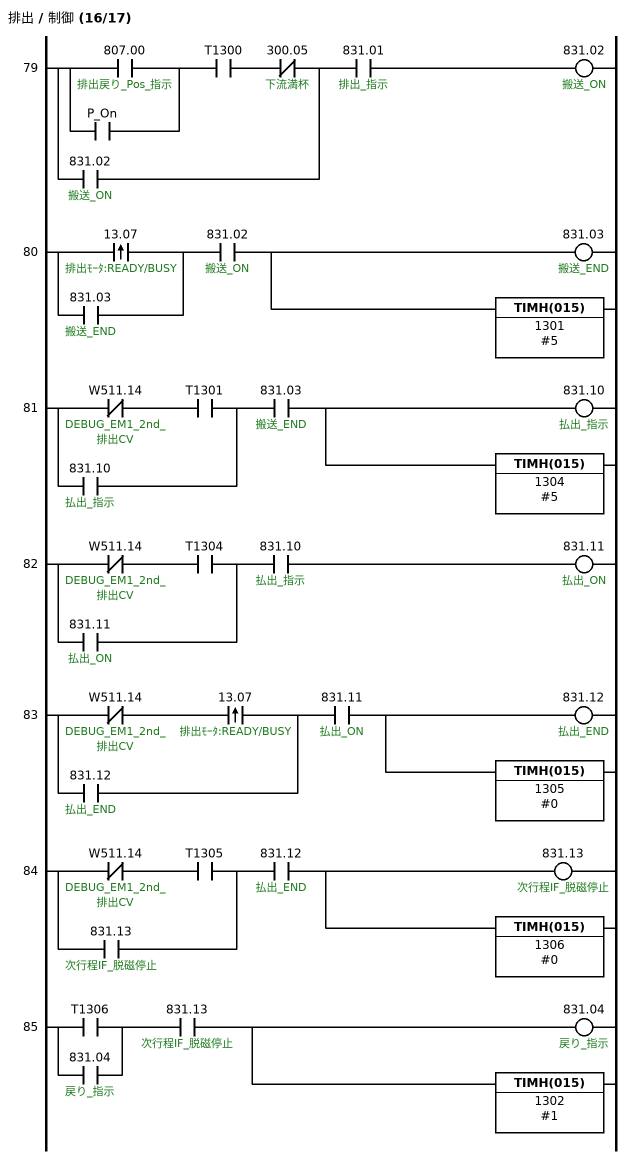
; [picture p192: 排出 / 制御, rungs 79-85]
; rung 79
LD 807.00  ; 排出戻り_Pos_指示
OR P_On
AND T1300
ANDNOT 300.05  ; 下流満杯
OR 831.02  ; 搬送_ON
AND 831.01  ; 排出_指示
OUT 831.02  ; 搬送_ON
; rung 80
@LD 13.07  ; 排出ﾓｰﾀ:READY/BUSY
OR 831.03  ; 搬送_END
AND 831.02  ; 搬送_ON
OUT 831.03  ; 搬送_END
TIMH(015) 1301 #5
; rung 81
LDNOT W511.14  ; DEBUG_EM1_2nd_排出CV
AND T1301
OR 831.10  ; 払出_指示
AND 831.03  ; 搬送_END
OUT 831.10  ; 払出_指示
TIMH(015) 1304 #5
; rung 82
LDNOT W511.14  ; DEBUG_EM1_2nd_排出CV
AND T1304
OR 831.11  ; 払出_ON
AND 831.10  ; 払出_指示
OUT 831.11  ; 払出_ON
; rung 83
LDNOT W511.14  ; DEBUG_EM1_2nd_排出CV
@AND 13.07  ; 排出ﾓｰﾀ:READY/BUSY
OR 831.12  ; 払出_END
AND 831.11  ; 払出_ON
OUT 831.12  ; 払出_END
TIMH(015) 1305 #0
; rung 84
LDNOT W511.14  ; DEBUG_EM1_2nd_排出CV
AND T1305
OR 831.13  ; 次行程IF_脱磁停止
AND 831.12  ; 払出_END
OUT 831.13  ; 次行程IF_脱磁停止
TIMH(015) 1306 #0
; rung 85
LD T1306
OR 831.04  ; 戻り_指示
AND 831.13  ; 次行程IF_脱磁停止
OUT 831.04  ; 戻り_指示
TIMH(015) 1302 #1

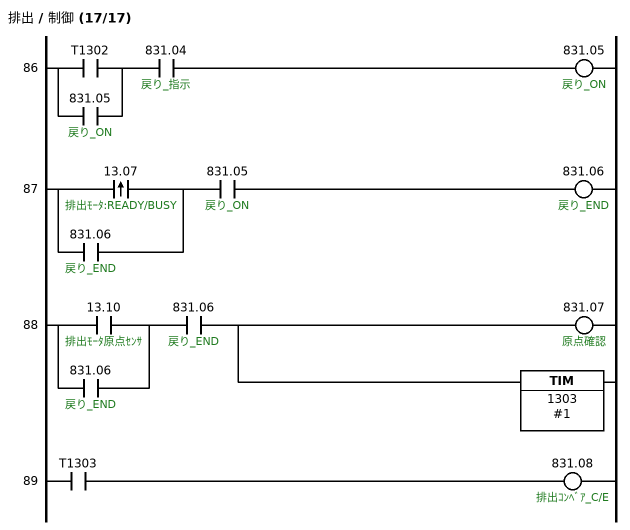
; rung 86
LD T1302
OR 831.05  ; 戻り_ON
AND 831.04  ; 戻り_指示
OUT 831.05  ; 戻り_ON
; rung 87
@LD 13.07  ; 排出ﾓｰﾀ:READY/BUSY
OR 831.06  ; 戻り_END
AND 831.05  ; 戻り_ON
OUT 831.06  ; 戻り_END
; rung 88
LD 13.10  ; 排出ﾓｰﾀ原点ｾﾝｻ
OR 831.06  ; 戻り_END
AND 831.06  ; 戻り_END
OUT 831.07  ; 原点確認
TIM 1303 #1
; rung 89
LD T1303
OUT 831.08  ; 排出ｺﾝﾍﾞｱ_C/E

### Section 出力

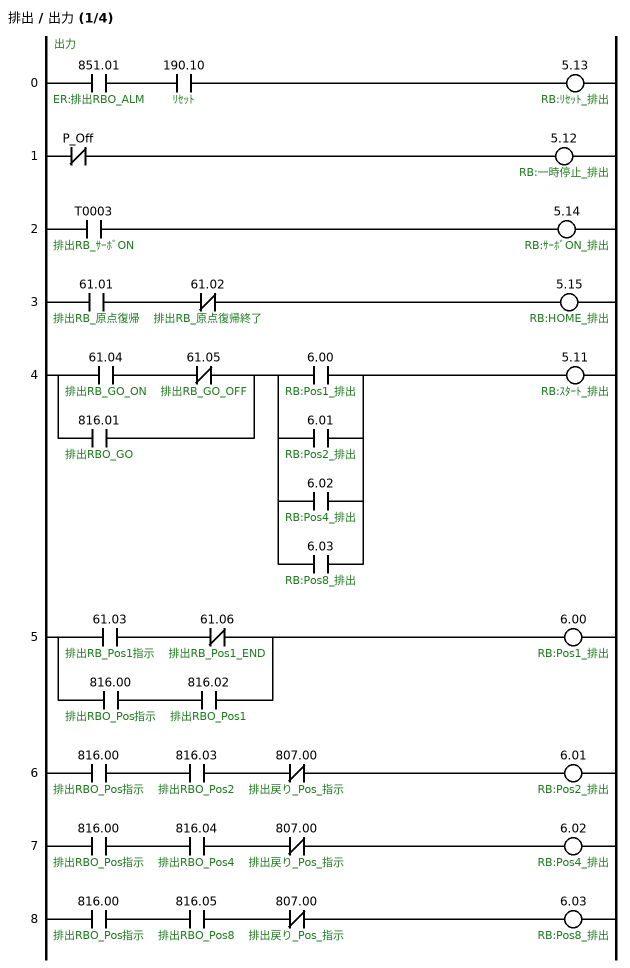
; rung 0: 出力
LD 851.01  ; ER:排出RBO_ALM
AND 190.10  ; ﾘｾｯﾄ
OUT 5.13  ; RB:ﾘｾｯﾄ_排出
; rung 1
LDNOT P_Off
OUT 5.12  ; RB:一時停止_排出
; rung 2
LD T0003  ; 排出RB_ｻｰﾎﾞON
OUT 5.14  ; RB:ｻｰﾎﾞON_排出
; rung 3
LD 61.01  ; 排出RB_原点復帰
ANDNOT 61.02  ; 排出RB_原点復帰終了
OUT 5.15  ; RB:HOME_排出
; rung 4
LD 61.04  ; 排出RB_GO_ON
ANDNOT 61.05  ; 排出RB_GO_OFF
OR 816.01  ; 排出RBO_GO
LD 6.00  ; RB:Pos1_排出
OR 6.01  ; RB:Pos2_排出
OR 6.02  ; RB:Pos4_排出
OR 6.03  ; RB:Pos8_排出
ANDLD
OUT 5.11  ; RB:ｽﾀｰﾄ_排出
; rung 5
LD 61.03  ; 排出RB_Pos1指示
ANDNOT 61.06  ; 排出RB_Pos1_END
LD 816.00  ; 排出RBO_Pos指示
AND 816.02  ; 排出RBO_Pos1
ORLD
OUT 6.00  ; RB:Pos1_排出
; rung 6
LD 816.00  ; 排出RBO_Pos指示
AND 816.03  ; 排出RBO_Pos2
ANDNOT 807.00  ; 排出戻り_Pos_指示
OUT 6.01  ; RB:Pos2_排出
; rung 7
LD 816.00  ; 排出RBO_Pos指示
AND 816.04  ; 排出RBO_Pos4
ANDNOT 807.00  ; 排出戻り_Pos_指示
OUT 6.02  ; RB:Pos4_排出
; rung 8
LD 816.00  ; 排出RBO_Pos指示
AND 816.05  ; 排出RBO_Pos8
ANDNOT 807.00  ; 排出戻り_Pos_指示
OUT 6.03  ; RB:Pos8_排出

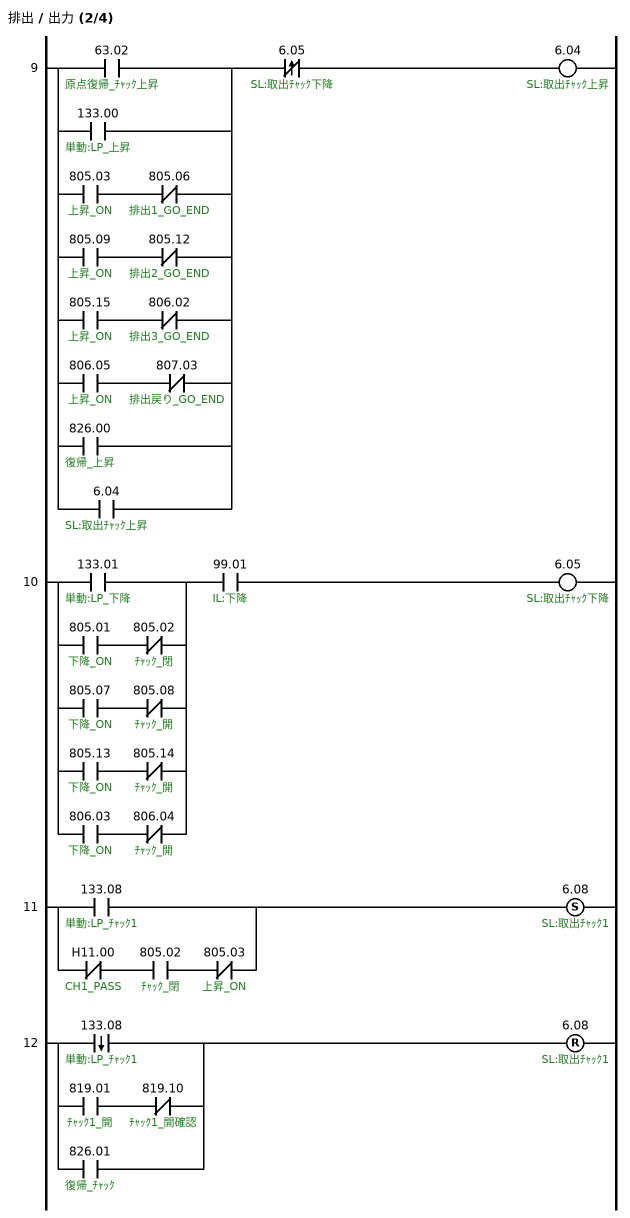
; rung 9
LD 63.02  ; 原点復帰_ﾁｬｯｸ上昇
OR 133.00  ; 単動:LP_上昇
LD 805.03  ; 上昇_ON
ANDNOT 805.06  ; 排出1_GO_END
ORLD
LD 805.09  ; 上昇_ON
ANDNOT 805.12  ; 排出2_GO_END
ORLD
LD 805.15  ; 上昇_ON
ANDNOT 806.02  ; 排出3_GO_END
ORLD
LD 806.05  ; 上昇_ON
ANDNOT 807.03  ; 排出戻り_GO_END
ORLD
OR 826.00  ; 復帰_上昇
OR 6.04  ; SL:取出ﾁｬｯｸ上昇
@ANDNOT 6.05  ; SL:取出ﾁｬｯｸ下降
OUT 6.04  ; SL:取出ﾁｬｯｸ上昇
; rung 10
LD 133.01  ; 単動:LP_下降
LD 805.01  ; 下降_ON
ANDNOT 805.02  ; ﾁｬｯｸ_閉
ORLD
LD 805.07  ; 下降_ON
ANDNOT 805.08  ; ﾁｬｯｸ_開
ORLD
LD 805.13  ; 下降_ON
ANDNOT 805.14  ; ﾁｬｯｸ_開
ORLD
LD 806.03  ; 下降_ON
ANDNOT 806.04  ; ﾁｬｯｸ_開
ORLD
AND 99.01  ; IL:下降
OUT 6.05  ; SL:取出ﾁｬｯｸ下降
; rung 11
LD 133.08  ; 単動:LP_ﾁｬｯｸ1
LDNOT H11.00  ; CH1_PASS
AND 805.02  ; ﾁｬｯｸ_閉
ANDNOT 805.03  ; 上昇_ON
ORLD
SET 6.08  ; SL:取出ﾁｬｯｸ1
; rung 12
%LD 133.08  ; 単動:LP_ﾁｬｯｸ1
LD 819.01  ; ﾁｬｯｸ1_開
ANDNOT 819.10  ; ﾁｬｯｸ1_開確認
ORLD
OR 826.01  ; 復帰_ﾁｬｯｸ
RSET 6.08  ; SL:取出ﾁｬｯｸ1

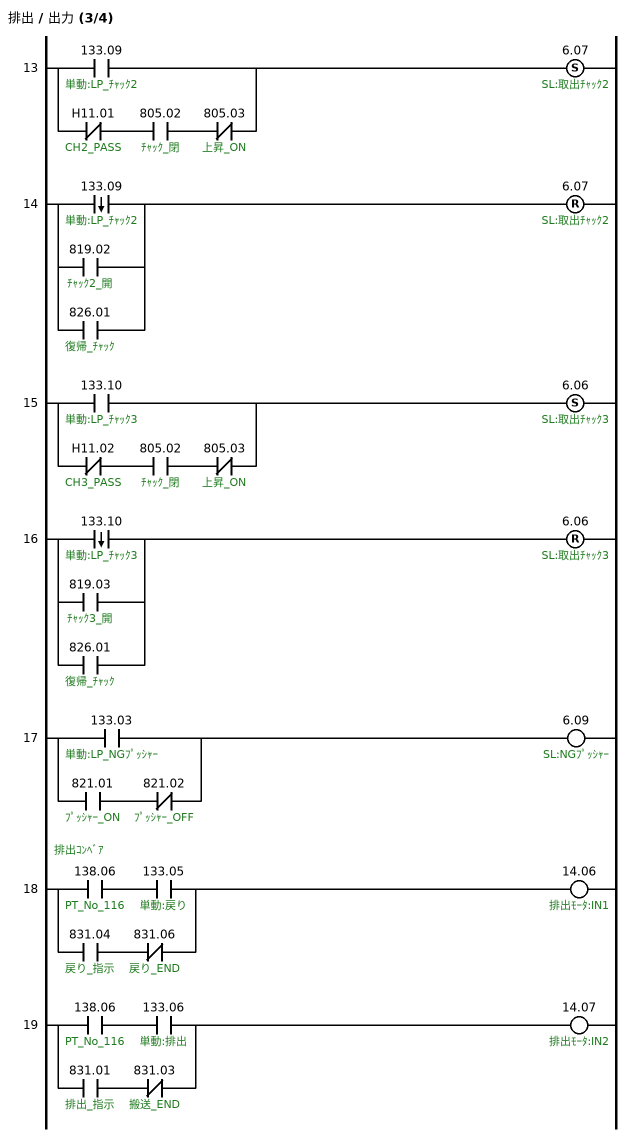
; rung 13
LD 133.09  ; 単動:LP_ﾁｬｯｸ2
LDNOT H11.01  ; CH2_PASS
AND 805.02  ; ﾁｬｯｸ_閉
ANDNOT 805.03  ; 上昇_ON
ORLD
SET 6.07  ; SL:取出ﾁｬｯｸ2
; rung 14
%LD 133.09  ; 単動:LP_ﾁｬｯｸ2
OR 819.02  ; ﾁｬｯｸ2_開
OR 826.01  ; 復帰_ﾁｬｯｸ
RSET 6.07  ; SL:取出ﾁｬｯｸ2
; rung 15
LD 133.10  ; 単動:LP_ﾁｬｯｸ3
LDNOT H11.02  ; CH3_PASS
AND 805.02  ; ﾁｬｯｸ_閉
ANDNOT 805.03  ; 上昇_ON
ORLD
SET 6.06  ; SL:取出ﾁｬｯｸ3
; rung 16
%LD 133.10  ; 単動:LP_ﾁｬｯｸ3
OR 819.03  ; ﾁｬｯｸ3_開
OR 826.01  ; 復帰_ﾁｬｯｸ
RSET 6.06  ; SL:取出ﾁｬｯｸ3
; rung 17
LD 133.03  ; 単動:LP_NGﾌﾟｯｼｬｰ
LD 821.01  ; ﾌﾟｯｼｬｰ_ON
ANDNOT 821.02  ; ﾌﾟｯｼｬｰ_OFF
ORLD
OUT 6.09  ; SL:NGﾌﾟｯｼｬｰ
; rung 18: 排出ｺﾝﾍﾞｱ
LD 138.06  ; PT_No_116
AND 133.05  ; 単動:戻り
LD 831.04  ; 戻り_指示
ANDNOT 831.06  ; 戻り_END
ORLD
OUT 14.06  ; 排出ﾓｰﾀ:IN1  // #1_戻り､#2_排出､#4_払出
; rung 19
LD 138.06  ; PT_No_116
AND 133.06  ; 単動:排出
LD 831.01  ; 排出_指示
ANDNOT 831.03  ; 搬送_END
ORLD
OUT 14.07  ; 排出ﾓｰﾀ:IN2

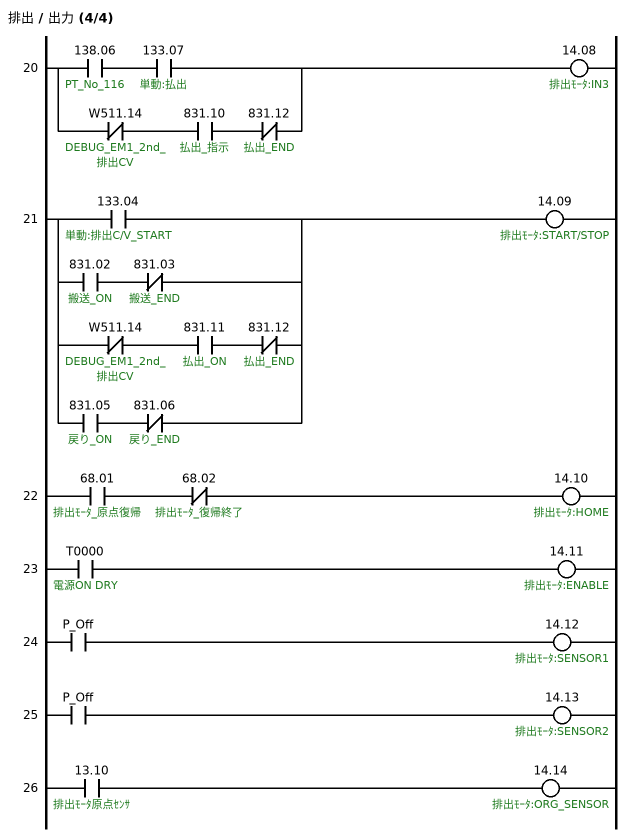
; rung 20
LD 138.06  ; PT_No_116
AND 133.07  ; 単動:払出
LDNOT W511.14  ; DEBUG_EM1_2nd_排出CV
AND 831.10  ; 払出_指示
ANDNOT 831.12  ; 払出_END
ORLD
OUT 14.08  ; 排出ﾓｰﾀ:IN3
; rung 21
LD 133.04  ; 単動:排出C/V_START
LD 831.02  ; 搬送_ON
ANDNOT 831.03  ; 搬送_END
ORLD
LDNOT W511.14  ; DEBUG_EM1_2nd_排出CV
AND 831.11  ; 払出_ON
ANDNOT 831.12  ; 払出_END
ORLD
LD 831.05  ; 戻り_ON
ANDNOT 831.06  ; 戻り_END
ORLD
OUT 14.09  ; 排出ﾓｰﾀ:START/STOP
; rung 22
LD 68.01  ; 排出ﾓｰﾀ_原点復帰
ANDNOT 68.02  ; 排出ﾓｰﾀ_復帰終了
OUT 14.10  ; 排出ﾓｰﾀ:HOME
; rung 23
LD T0000  ; 電源ON DRY
OUT 14.11  ; 排出ﾓｰﾀ:ENABLE
; rung 24
LD P_Off
OUT 14.12  ; 排出ﾓｰﾀ:SENSOR1
; rung 25
LD P_Off
OUT 14.13  ; 排出ﾓｰﾀ:SENSOR2
; rung 26
LD 13.10  ; 排出ﾓｰﾀ原点ｾﾝｻ
OUT 14.14  ; 排出ﾓｰﾀ:ORG_SENSOR

### Section ｴﾗｰ

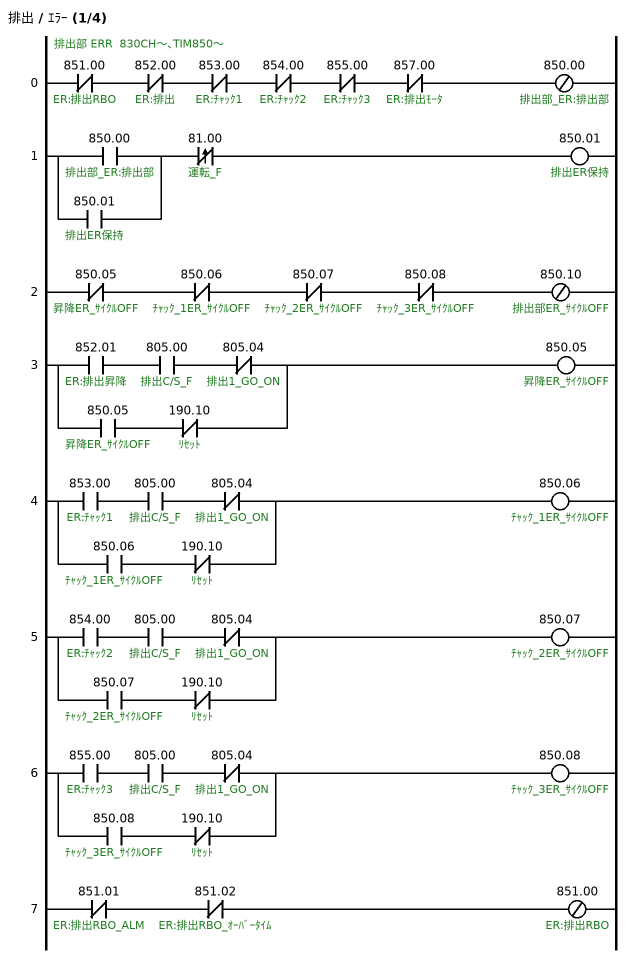
; rung 0: 排出部 ERR  830CH～､TIM850～
LDNOT 851.00  ; ER:排出RBO
ANDNOT 852.00  ; ER:排出
ANDNOT 853.00  ; ER:ﾁｬｯｸ1
ANDNOT 854.00  ; ER:ﾁｬｯｸ2
ANDNOT 855.00  ; ER:ﾁｬｯｸ3
ANDNOT 857.00  ; ER:排出ﾓｰﾀ
OUTNOT 850.00  ; 排出部_ER:排出部
; rung 1
LD 850.00  ; 排出部_ER:排出部
OR 850.01  ; 排出ER保持
@ANDNOT 81.00  ; 運転_F
OUT 850.01  ; 排出ER保持
; rung 2
LDNOT 850.05  ; 昇降ER_ｻｲｸﾙOFF
ANDNOT 850.06  ; ﾁｬｯｸ_1ER_ｻｲｸﾙOFF
ANDNOT 850.07  ; ﾁｬｯｸ_2ER_ｻｲｸﾙOFF
ANDNOT 850.08  ; ﾁｬｯｸ_3ER_ｻｲｸﾙOFF
OUTNOT 850.10  ; 排出部ER_ｻｲｸﾙOFF
; rung 3
LD 852.01  ; ER:排出昇降
AND 805.00  ; 排出C/S_F
ANDNOT 805.04  ; 排出1_GO_ON
LD 850.05  ; 昇降ER_ｻｲｸﾙOFF
ANDNOT 190.10  ; ﾘｾｯﾄ
ORLD
OUT 850.05  ; 昇降ER_ｻｲｸﾙOFF
; rung 4
LD 853.00  ; ER:ﾁｬｯｸ1
AND 805.00  ; 排出C/S_F
ANDNOT 805.04  ; 排出1_GO_ON
LD 850.06  ; ﾁｬｯｸ_1ER_ｻｲｸﾙOFF
ANDNOT 190.10  ; ﾘｾｯﾄ
ORLD
OUT 850.06  ; ﾁｬｯｸ_1ER_ｻｲｸﾙOFF
; rung 5
LD 854.00  ; ER:ﾁｬｯｸ2
AND 805.00  ; 排出C/S_F
ANDNOT 805.04  ; 排出1_GO_ON
LD 850.07  ; ﾁｬｯｸ_2ER_ｻｲｸﾙOFF
ANDNOT 190.10  ; ﾘｾｯﾄ
ORLD
OUT 850.07  ; ﾁｬｯｸ_2ER_ｻｲｸﾙOFF
; rung 6
LD 855.00  ; ER:ﾁｬｯｸ3
AND 805.00  ; 排出C/S_F
ANDNOT 805.04  ; 排出1_GO_ON
LD 850.08  ; ﾁｬｯｸ_3ER_ｻｲｸﾙOFF
ANDNOT 190.10  ; ﾘｾｯﾄ
ORLD
OUT 850.08  ; ﾁｬｯｸ_3ER_ｻｲｸﾙOFF
; rung 7
LDNOT 851.01  ; ER:排出RBO_ALM
ANDNOT 851.02  ; ER:排出RBO_ｵｰﾊﾞｰﾀｲﾑ
OUTNOT 851.00  ; ER:排出RBO

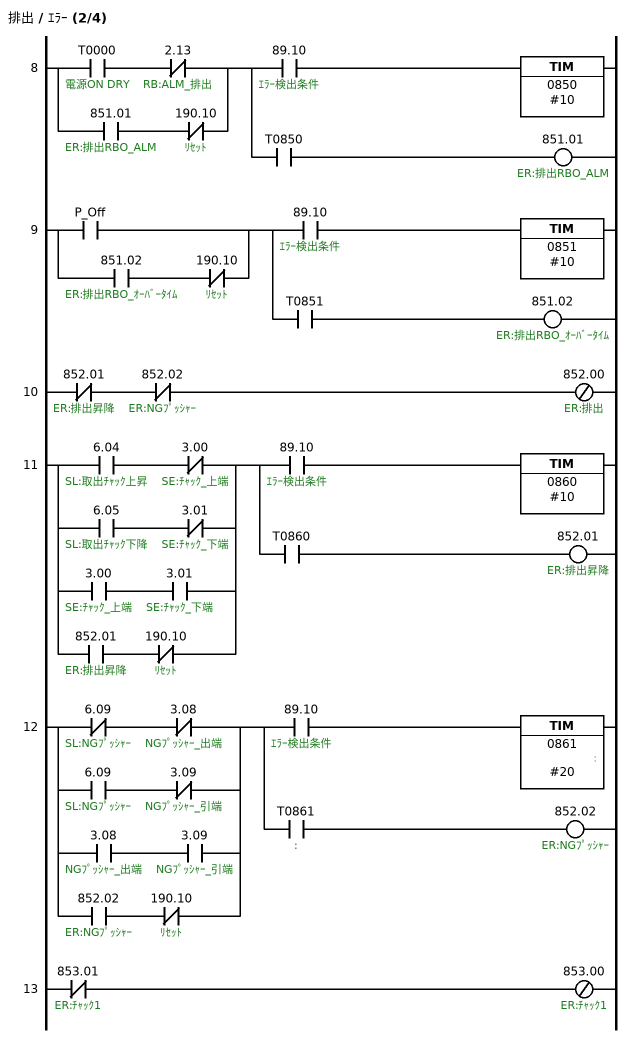
; rung 8
LD T0000  ; 電源ON DRY
ANDNOT 2.13  ; RB:ALM_排出
LD 851.01  ; ER:排出RBO_ALM
ANDNOT 190.10  ; ﾘｾｯﾄ
ORLD
OUT TR0
AND 89.10  ; ｴﾗｰ検出条件
TIM 0850 #10
LD TR0
AND T0850
OUT 851.01  ; ER:排出RBO_ALM
; rung 9
LD P_Off
LD 851.02  ; ER:排出RBO_ｵｰﾊﾞｰﾀｲﾑ
ANDNOT 190.10  ; ﾘｾｯﾄ
ORLD
OUT TR0
AND 89.10  ; ｴﾗｰ検出条件
TIM 0851 #10
LD TR0
AND T0851
OUT 851.02  ; ER:排出RBO_ｵｰﾊﾞｰﾀｲﾑ
; rung 10
LDNOT 852.01  ; ER:排出昇降
ANDNOT 852.02  ; ER:NGﾌﾟｯｼｬｰ
OUTNOT 852.00  ; ER:排出
; rung 11
LD 6.04  ; SL:取出ﾁｬｯｸ上昇
ANDNOT 3.00  ; SE:ﾁｬｯｸ_上端
LD 6.05  ; SL:取出ﾁｬｯｸ下降
ANDNOT 3.01  ; SE:ﾁｬｯｸ_下端
ORLD
LD 3.00  ; SE:ﾁｬｯｸ_上端
AND 3.01  ; SE:ﾁｬｯｸ_下端
ORLD
LD 852.01  ; ER:排出昇降
ANDNOT 190.10  ; ﾘｾｯﾄ
ORLD
OUT TR0
AND 89.10  ; ｴﾗｰ検出条件
TIM 0860 #10
LD TR0
AND T0860
OUT 852.01  ; ER:排出昇降
; rung 12
LDNOT 6.09  ; SL:NGﾌﾟｯｼｬｰ
ANDNOT 3.08  ; NGﾌﾟｯｼｬｰ_出端
LD 6.09  ; SL:NGﾌﾟｯｼｬｰ
ANDNOT 3.09  ; NGﾌﾟｯｼｬｰ_引端
ORLD
LD 3.08  ; NGﾌﾟｯｼｬｰ_出端
AND 3.09  ; NGﾌﾟｯｼｬｰ_引端
ORLD
LD 852.02  ; ER:NGﾌﾟｯｼｬｰ
ANDNOT 190.10  ; ﾘｾｯﾄ
ORLD
OUT TR0
AND 89.10  ; ｴﾗｰ検出条件
TIM 0861 #20  ; :
LD TR0
AND T0861  ; :
OUT 852.02  ; ER:NGﾌﾟｯｼｬｰ
; rung 13
LDNOT 853.01  ; ER:ﾁｬｯｸ1
OUTNOT 853.00  ; ER:ﾁｬｯｸ1

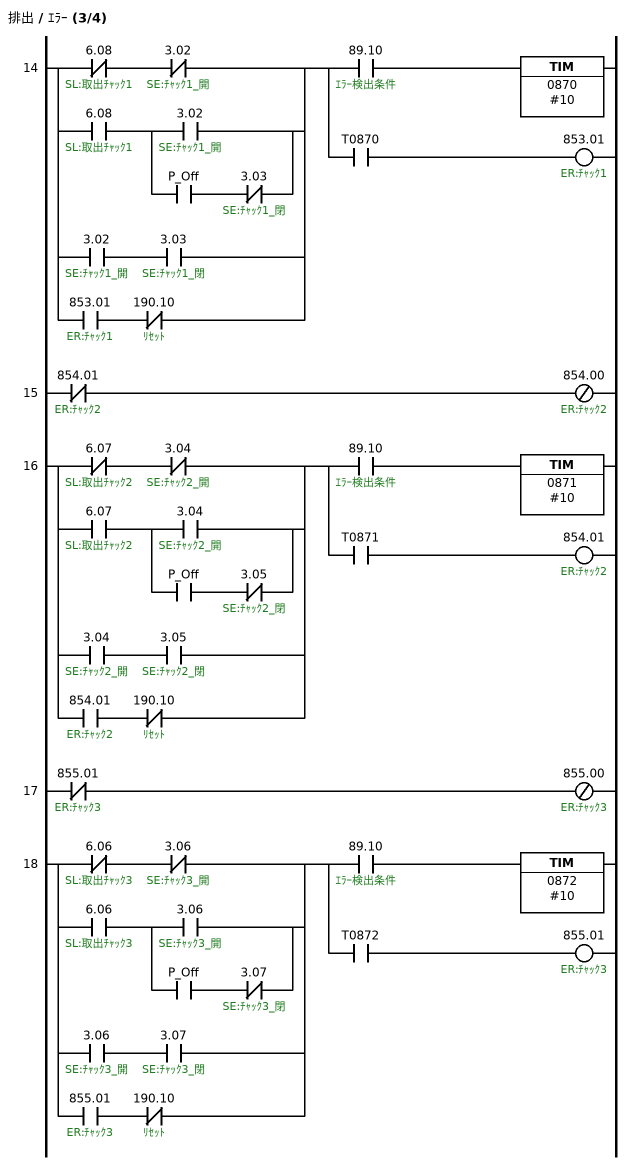
; rung 14
LDNOT 6.08  ; SL:取出ﾁｬｯｸ1
ANDNOT 3.02  ; SE:ﾁｬｯｸ1_開
LD 6.08  ; SL:取出ﾁｬｯｸ1
LD 3.02  ; SE:ﾁｬｯｸ1_開
LD P_Off
ANDNOT 3.03  ; SE:ﾁｬｯｸ1_閉
ORLD
ANDLD
ORLD
LD 3.02  ; SE:ﾁｬｯｸ1_開
AND 3.03  ; SE:ﾁｬｯｸ1_閉
ORLD
LD 853.01  ; ER:ﾁｬｯｸ1
ANDNOT 190.10  ; ﾘｾｯﾄ
ORLD
OUT TR0
AND 89.10  ; ｴﾗｰ検出条件
TIM 0870 #10
LD TR0
AND T0870
OUT 853.01  ; ER:ﾁｬｯｸ1
; rung 15
LDNOT 854.01  ; ER:ﾁｬｯｸ2
OUTNOT 854.00  ; ER:ﾁｬｯｸ2
; rung 16
LDNOT 6.07  ; SL:取出ﾁｬｯｸ2
ANDNOT 3.04  ; SE:ﾁｬｯｸ2_開
LD 6.07  ; SL:取出ﾁｬｯｸ2
LD 3.04  ; SE:ﾁｬｯｸ2_開
LD P_Off
ANDNOT 3.05  ; SE:ﾁｬｯｸ2_閉
ORLD
ANDLD
ORLD
LD 3.04  ; SE:ﾁｬｯｸ2_開
AND 3.05  ; SE:ﾁｬｯｸ2_閉
ORLD
LD 854.01  ; ER:ﾁｬｯｸ2
ANDNOT 190.10  ; ﾘｾｯﾄ
ORLD
OUT TR0
AND 89.10  ; ｴﾗｰ検出条件
TIM 0871 #10
LD TR0
AND T0871
OUT 854.01  ; ER:ﾁｬｯｸ2
; rung 17
LDNOT 855.01  ; ER:ﾁｬｯｸ3
OUTNOT 855.00  ; ER:ﾁｬｯｸ3
; rung 18
LDNOT 6.06  ; SL:取出ﾁｬｯｸ3
ANDNOT 3.06  ; SE:ﾁｬｯｸ3_開
LD 6.06  ; SL:取出ﾁｬｯｸ3
LD 3.06  ; SE:ﾁｬｯｸ3_開
LD P_Off
ANDNOT 3.07  ; SE:ﾁｬｯｸ3_閉
ORLD
ANDLD
ORLD
LD 3.06  ; SE:ﾁｬｯｸ3_開
AND 3.07  ; SE:ﾁｬｯｸ3_閉
ORLD
LD 855.01  ; ER:ﾁｬｯｸ3
ANDNOT 190.10  ; ﾘｾｯﾄ
ORLD
OUT TR0
AND 89.10  ; ｴﾗｰ検出条件
TIM 0872 #10
LD TR0
AND T0872
OUT 855.01  ; ER:ﾁｬｯｸ3

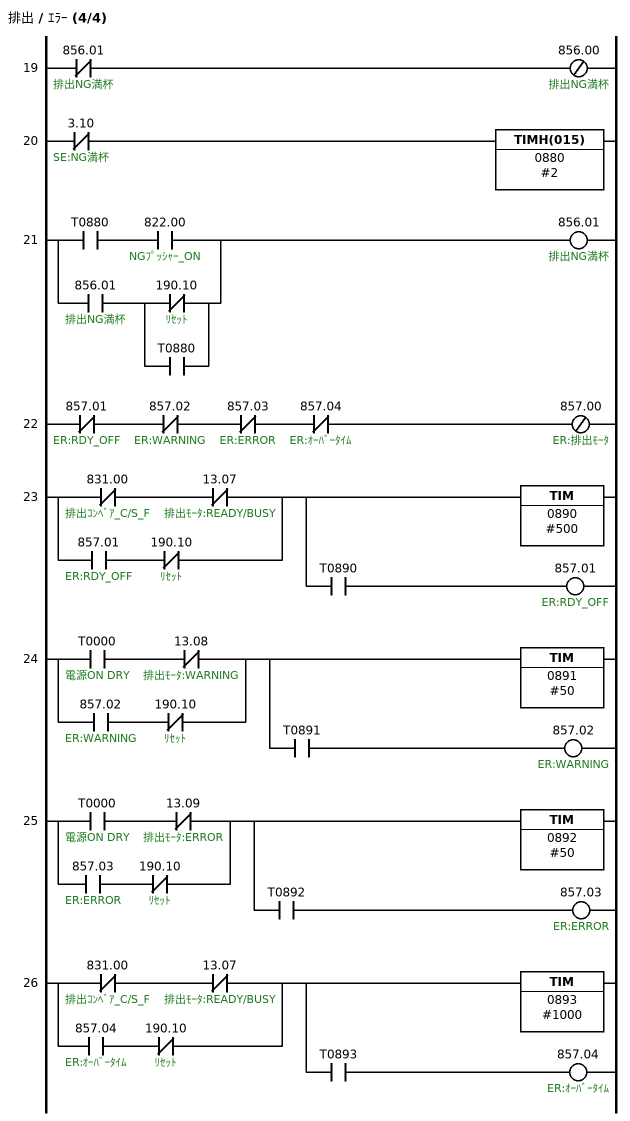
; rung 19
LDNOT 856.01  ; 排出NG満杯
OUTNOT 856.00  ; 排出NG満杯
; rung 20
LDNOT 3.10  ; SE:NG満杯
TIMH(015) 0880 #2
; rung 21
LD T0880
AND 822.00  ; NGﾌﾟｯｼｬｰ_ON
LD 856.01  ; 排出NG満杯
LDNOT 190.10  ; ﾘｾｯﾄ
OR T0880
ANDLD
ORLD
OUT 856.01  ; 排出NG満杯
; rung 22
LDNOT 857.01  ; ER:RDY_OFF
ANDNOT 857.02  ; ER:WARNING
ANDNOT 857.03  ; ER:ERROR
ANDNOT 857.04  ; ER:ｵｰﾊﾞｰﾀｲﾑ
OUTNOT 857.00  ; ER:排出ﾓｰﾀ
; rung 23
LDNOT 831.00  ; 排出ｺﾝﾍﾞｱ_C/S_F
ANDNOT 13.07  ; 排出ﾓｰﾀ:READY/BUSY
LD 857.01  ; ER:RDY_OFF
ANDNOT 190.10  ; ﾘｾｯﾄ
ORLD
TIM 0890 #500
AND T0890
OUT 857.01  ; ER:RDY_OFF
; rung 24
LD T0000  ; 電源ON DRY
ANDNOT 13.08  ; 排出ﾓｰﾀ:WARNING
LD 857.02  ; ER:WARNING
ANDNOT 190.10  ; ﾘｾｯﾄ
ORLD
TIM 0891 #50
AND T0891
OUT 857.02  ; ER:WARNING
; rung 25
LD T0000  ; 電源ON DRY
ANDNOT 13.09  ; 排出ﾓｰﾀ:ERROR
LD 857.03  ; ER:ERROR
ANDNOT 190.10  ; ﾘｾｯﾄ
ORLD
TIM 0892 #50
AND T0892
OUT 857.03  ; ER:ERROR
; rung 26
LDNOT 831.00  ; 排出ｺﾝﾍﾞｱ_C/S_F
ANDNOT 13.07  ; 排出ﾓｰﾀ:READY/BUSY
LD 857.04  ; ER:ｵｰﾊﾞｰﾀｲﾑ
ANDNOT 190.10  ; ﾘｾｯﾄ
ORLD
TIM 0893 #1000
AND T0893
OUT 857.04  ; ER:ｵｰﾊﾞｰﾀｲﾑ

### Section END
; rung 0
END(001)

## Program ﾃﾞｰﾀ収集 (cyclic task 9)

### Section 通信ST

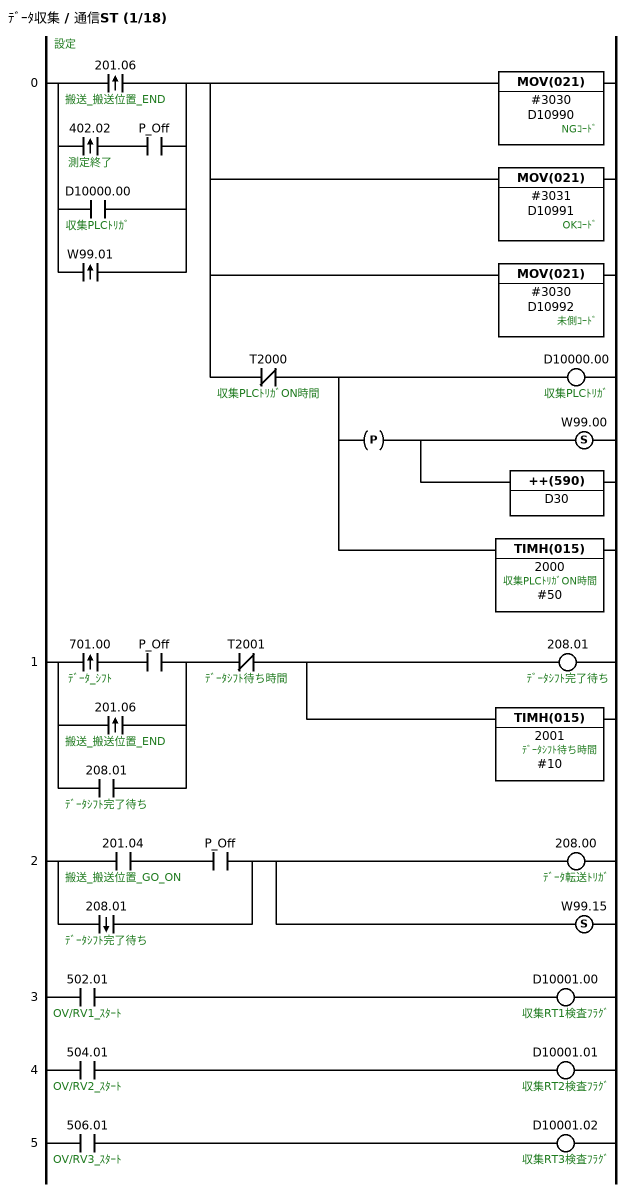
; rung 0: 設定
@LD 201.06  ; 搬送_搬送位置_END
@LD 402.02  ; 測定終了
AND P_Off
ORLD
OR D10000.00  ; 収集PLCﾄﾘｶﾞ
@OR W99.01
MOV(021) #3030 D10990  ; NGｺｰﾄﾞ
MOV(021) #3031 D10991  ; OKｺｰﾄﾞ
MOV(021) #3030 D10992  ; 未側ｺｰﾄﾞ
ANDNOT T2000  ; 収集PLCﾄﾘｶﾞON時間
OUT TR0
OUT D10000.00  ; 収集PLCﾄﾘｶﾞ
UP(521)
SET W99.00
++(590) D30
LD TR0
TIMH(015) 2000 #50  ; 収集PLCﾄﾘｶﾞON時間
; rung 1
@LD 701.00  ; ﾃﾞｰﾀ_ｼﾌﾄ
AND P_Off
@OR 201.06  ; 搬送_搬送位置_END
OR 208.01  ; ﾃﾞｰﾀｼﾌﾄ完了待ち
ANDNOT T2001  ; ﾃﾞｰﾀｼﾌﾄ待ち時間
OUT 208.01  ; ﾃﾞｰﾀｼﾌﾄ完了待ち
TIMH(015) 2001 #10  ; ﾃﾞｰﾀｼﾌﾄ待ち時間
; rung 2
LD 201.04  ; 搬送_搬送位置_GO_ON
AND P_Off
%OR 208.01  ; ﾃﾞｰﾀｼﾌﾄ完了待ち
OUT 208.00  ; ﾃﾞｰﾀ転送ﾄﾘｶﾞ
SET W99.15
; rung 3
LD 502.01  ; OV/RV1_ｽﾀｰﾄ
OUT D10001.00  ; 収集RT1検査ﾌﾗｸﾞ
; rung 4
LD 504.01  ; OV/RV2_ｽﾀｰﾄ
OUT D10001.01  ; 収集RT2検査ﾌﾗｸﾞ
; rung 5
LD 506.01  ; OV/RV3_ｽﾀｰﾄ
OUT D10001.02  ; 収集RT3検査ﾌﾗｸﾞ

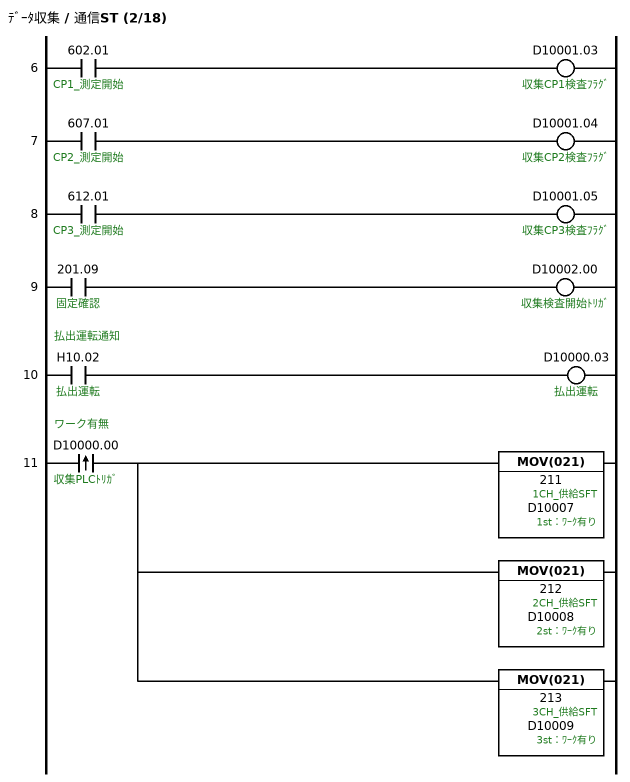
; rung 6
LD 602.01  ; CP1_測定開始
OUT D10001.03  ; 収集CP1検査ﾌﾗｸﾞ
; rung 7
LD 607.01  ; CP2_測定開始
OUT D10001.04  ; 収集CP2検査ﾌﾗｸﾞ
; rung 8
LD 612.01  ; CP3_測定開始
OUT D10001.05  ; 収集CP3検査ﾌﾗｸﾞ
; rung 9
LD 201.09  ; 固定確認
OUT D10002.00  ; 収集検査開始ﾄﾘｶﾞ
; rung 10: 払出運転通知
LD H10.02  ; 払出運転
OUT D10000.03  ; 払出運転
; rung 11: ワーク有無
@LD D10000.00  ; 収集PLCﾄﾘｶﾞ
MOV(021) 211 D10007  ; 1CH_供給SFT, 1st：ﾜｰｸ有り
MOV(021) 212 D10008  ; 2CH_供給SFT, 2st：ﾜｰｸ有り
MOV(021) 213 D10009  ; 3CH_供給SFT, 3st：ﾜｰｸ有り

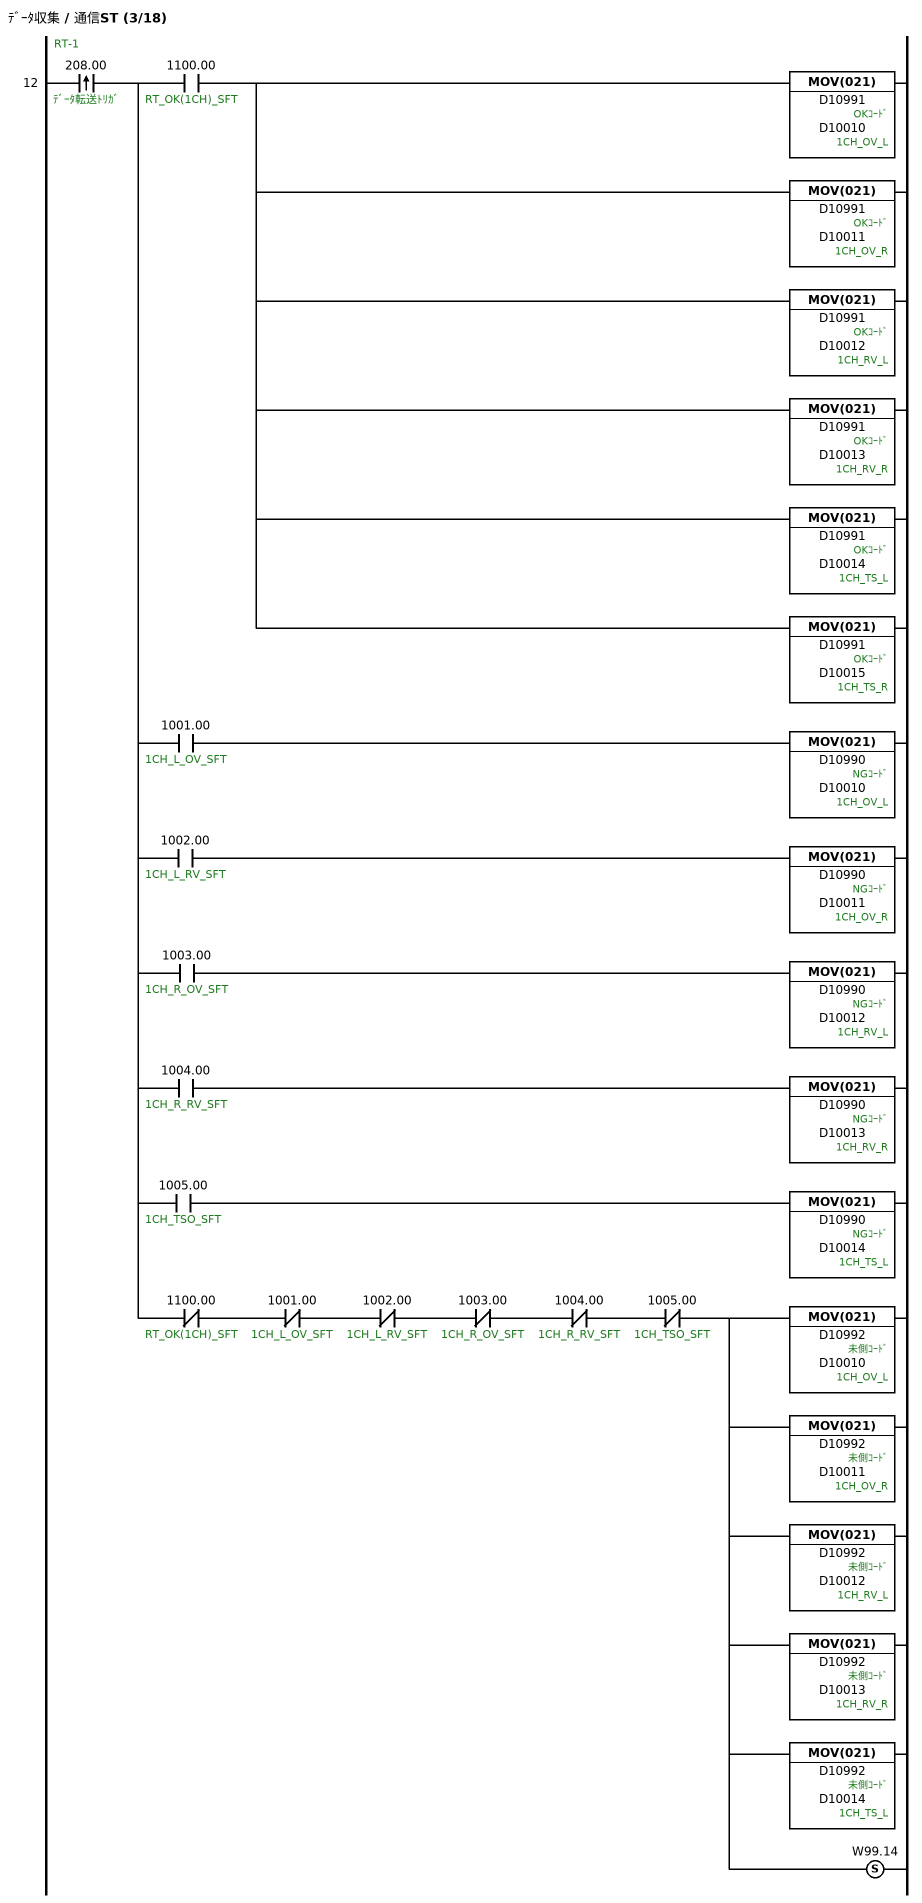
; rung 12: RT-1
@LD 208.00  ; ﾃﾞｰﾀ転送ﾄﾘｶﾞ
OUT TR0
AND 1100.00  ; RT_OK(1CH)_SFT
MOV(021) D10991 D10010  ; OKｺｰﾄﾞ, 1CH_OV_L
MOV(021) D10991 D10011  ; OKｺｰﾄﾞ, 1CH_OV_R
MOV(021) D10991 D10012  ; OKｺｰﾄﾞ, 1CH_RV_L
MOV(021) D10991 D10013  ; OKｺｰﾄﾞ, 1CH_RV_R
MOV(021) D10991 D10014  ; OKｺｰﾄﾞ, 1CH_TS_L
MOV(021) D10991 D10015  ; OKｺｰﾄﾞ, 1CH_TS_R
LD TR0
AND 1001.00  ; 1CH_L_OV_SFT
MOV(021) D10990 D10010  ; NGｺｰﾄﾞ, 1CH_OV_L
LD TR0
AND 1002.00  ; 1CH_L_RV_SFT
MOV(021) D10990 D10011  ; NGｺｰﾄﾞ, 1CH_OV_R
LD TR0
AND 1003.00  ; 1CH_R_OV_SFT
MOV(021) D10990 D10012  ; NGｺｰﾄﾞ, 1CH_RV_L
LD TR0
AND 1004.00  ; 1CH_R_RV_SFT
MOV(021) D10990 D10013  ; NGｺｰﾄﾞ, 1CH_RV_R
LD TR0
AND 1005.00  ; 1CH_TSO_SFT
MOV(021) D10990 D10014  ; NGｺｰﾄﾞ, 1CH_TS_L
LD TR0
ANDNOT 1100.00  ; RT_OK(1CH)_SFT
ANDNOT 1001.00  ; 1CH_L_OV_SFT
ANDNOT 1002.00  ; 1CH_L_RV_SFT
ANDNOT 1003.00  ; 1CH_R_OV_SFT
ANDNOT 1004.00  ; 1CH_R_RV_SFT
ANDNOT 1005.00  ; 1CH_TSO_SFT
MOV(021) D10992 D10010  ; 未側ｺｰﾄﾞ, 1CH_OV_L
MOV(021) D10992 D10011  ; 未側ｺｰﾄﾞ, 1CH_OV_R
MOV(021) D10992 D10012  ; 未側ｺｰﾄﾞ, 1CH_RV_L
MOV(021) D10992 D10013  ; 未側ｺｰﾄﾞ, 1CH_RV_R
MOV(021) D10992 D10014  ; 未側ｺｰﾄﾞ, 1CH_TS_L
SET W99.14

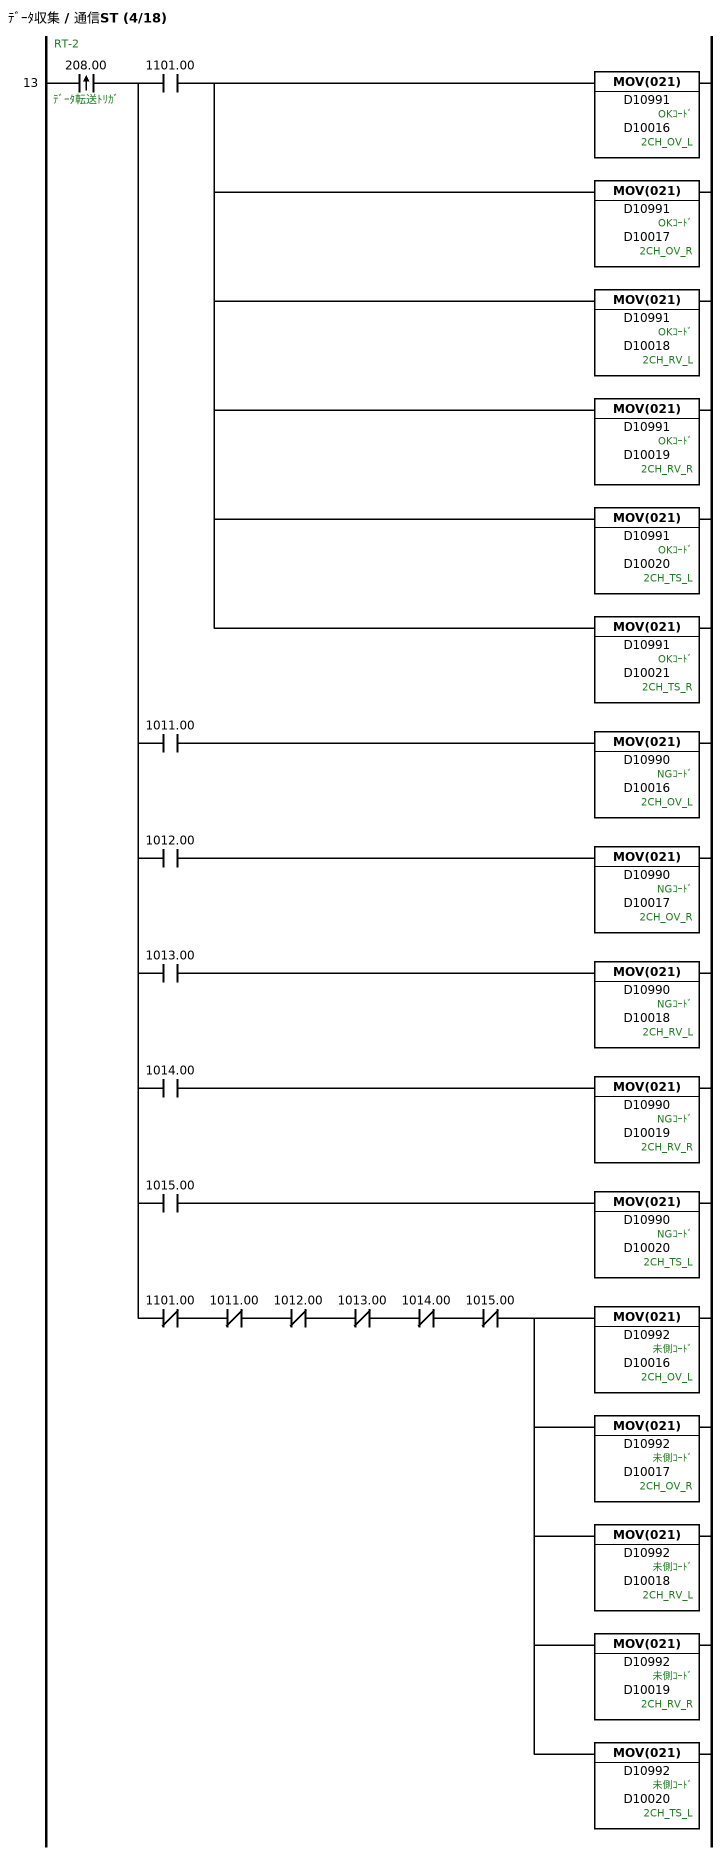
; rung 13: RT-2
@LD 208.00  ; ﾃﾞｰﾀ転送ﾄﾘｶﾞ
OUT TR0
AND 1101.00
MOV(021) D10991 D10016  ; OKｺｰﾄﾞ, 2CH_OV_L
MOV(021) D10991 D10017  ; OKｺｰﾄﾞ, 2CH_OV_R
MOV(021) D10991 D10018  ; OKｺｰﾄﾞ, 2CH_RV_L
MOV(021) D10991 D10019  ; OKｺｰﾄﾞ, 2CH_RV_R
MOV(021) D10991 D10020  ; OKｺｰﾄﾞ, 2CH_TS_L
MOV(021) D10991 D10021  ; OKｺｰﾄﾞ, 2CH_TS_R
LD TR0
AND 1011.00
MOV(021) D10990 D10016  ; NGｺｰﾄﾞ, 2CH_OV_L
LD TR0
AND 1012.00
MOV(021) D10990 D10017  ; NGｺｰﾄﾞ, 2CH_OV_R
LD TR0
AND 1013.00
MOV(021) D10990 D10018  ; NGｺｰﾄﾞ, 2CH_RV_L
LD TR0
AND 1014.00
MOV(021) D10990 D10019  ; NGｺｰﾄﾞ, 2CH_RV_R
LD TR0
AND 1015.00
MOV(021) D10990 D10020  ; NGｺｰﾄﾞ, 2CH_TS_L
LD TR0
ANDNOT 1101.00
ANDNOT 1011.00
ANDNOT 1012.00
ANDNOT 1013.00
ANDNOT 1014.00
ANDNOT 1015.00
MOV(021) D10992 D10016  ; 未側ｺｰﾄﾞ, 2CH_OV_L
MOV(021) D10992 D10017  ; 未側ｺｰﾄﾞ, 2CH_OV_R
MOV(021) D10992 D10018  ; 未側ｺｰﾄﾞ, 2CH_RV_L
MOV(021) D10992 D10019  ; 未側ｺｰﾄﾞ, 2CH_RV_R
MOV(021) D10992 D10020  ; 未側ｺｰﾄﾞ, 2CH_TS_L

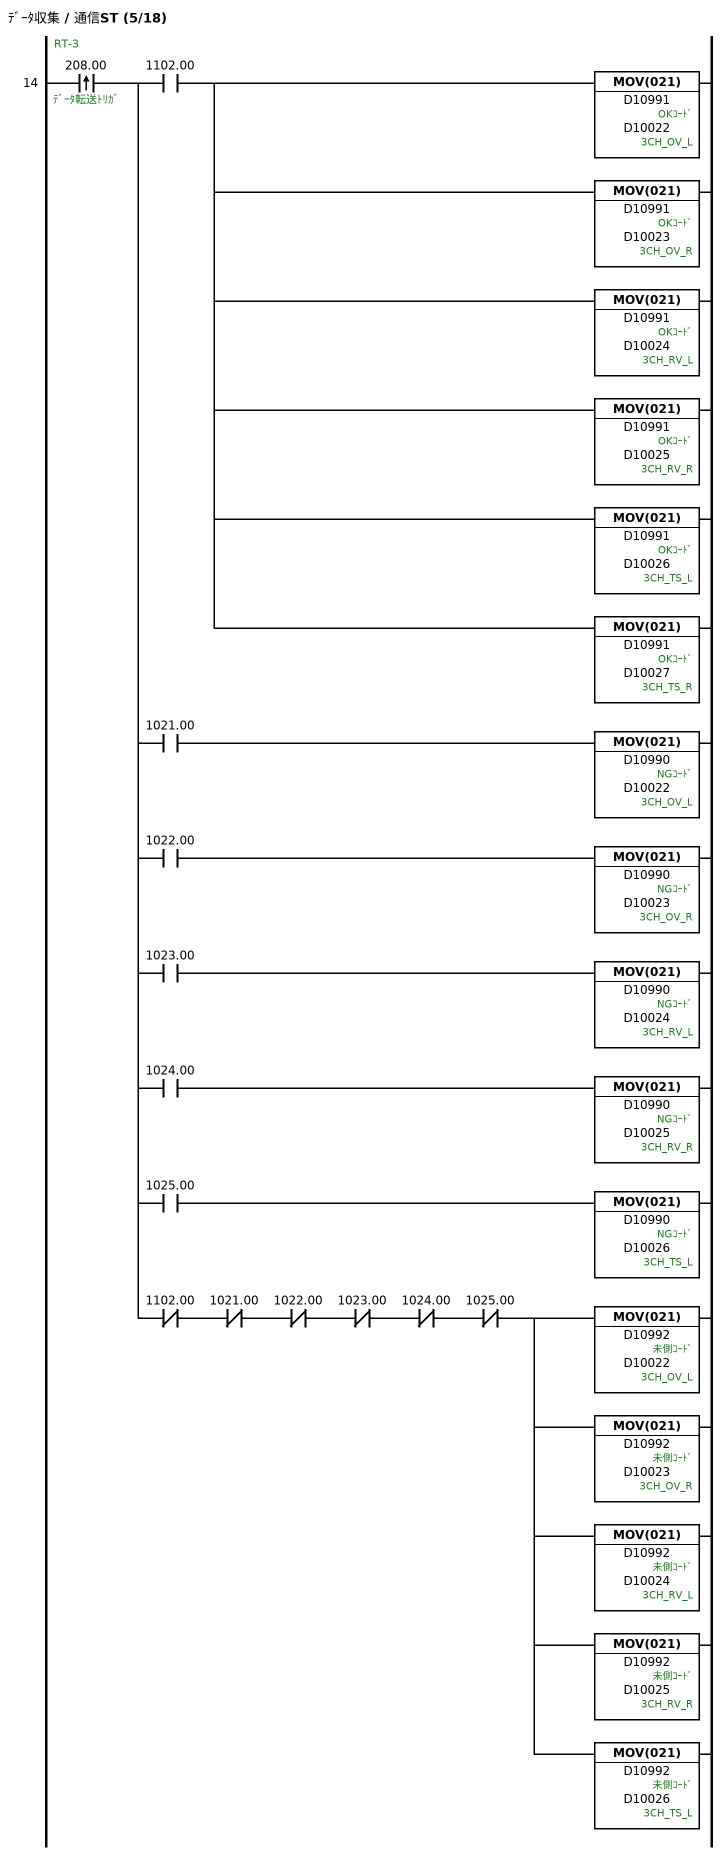
; rung 14: RT-3
@LD 208.00  ; ﾃﾞｰﾀ転送ﾄﾘｶﾞ
OUT TR0
AND 1102.00
MOV(021) D10991 D10022  ; OKｺｰﾄﾞ, 3CH_OV_L
MOV(021) D10991 D10023  ; OKｺｰﾄﾞ, 3CH_OV_R
MOV(021) D10991 D10024  ; OKｺｰﾄﾞ, 3CH_RV_L
MOV(021) D10991 D10025  ; OKｺｰﾄﾞ, 3CH_RV_R
MOV(021) D10991 D10026  ; OKｺｰﾄﾞ, 3CH_TS_L
MOV(021) D10991 D10027  ; OKｺｰﾄﾞ, 3CH_TS_R
LD TR0
AND 1021.00
MOV(021) D10990 D10022  ; NGｺｰﾄﾞ, 3CH_OV_L
LD TR0
AND 1022.00
MOV(021) D10990 D10023  ; NGｺｰﾄﾞ, 3CH_OV_R
LD TR0
AND 1023.00
MOV(021) D10990 D10024  ; NGｺｰﾄﾞ, 3CH_RV_L
LD TR0
AND 1024.00
MOV(021) D10990 D10025  ; NGｺｰﾄﾞ, 3CH_RV_R
LD TR0
AND 1025.00
MOV(021) D10990 D10026  ; NGｺｰﾄﾞ, 3CH_TS_L
LD TR0
ANDNOT 1102.00
ANDNOT 1021.00
ANDNOT 1022.00
ANDNOT 1023.00
ANDNOT 1024.00
ANDNOT 1025.00
MOV(021) D10992 D10022  ; 未側ｺｰﾄﾞ, 3CH_OV_L
MOV(021) D10992 D10023  ; 未側ｺｰﾄﾞ, 3CH_OV_R
MOV(021) D10992 D10024  ; 未側ｺｰﾄﾞ, 3CH_RV_L
MOV(021) D10992 D10025  ; 未側ｺｰﾄﾞ, 3CH_RV_R
MOV(021) D10992 D10026  ; 未側ｺｰﾄﾞ, 3CH_TS_L

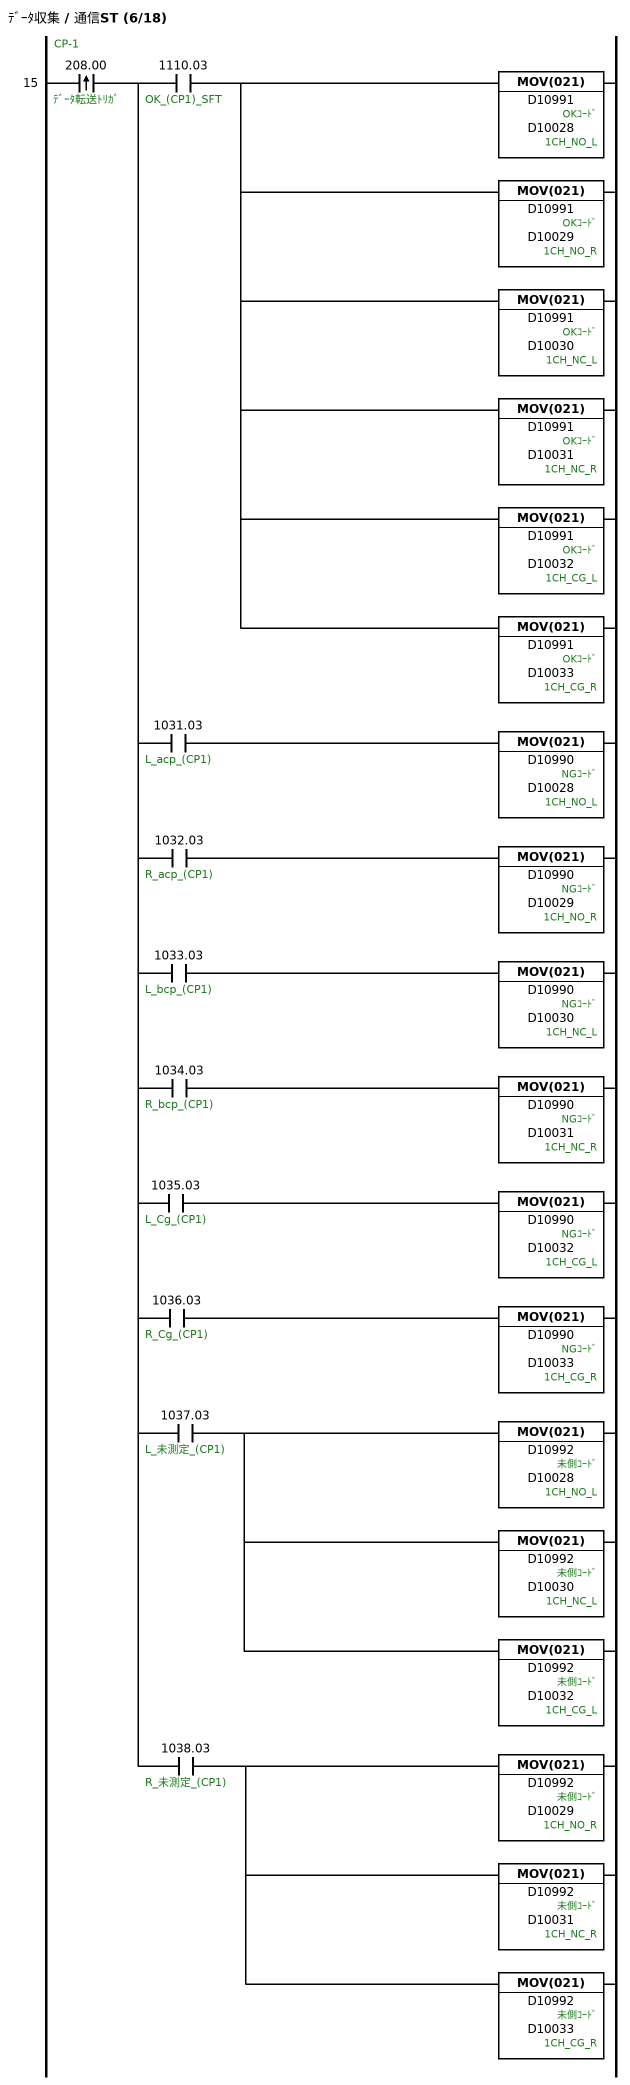
; rung 15: CP-1
@LD 208.00  ; ﾃﾞｰﾀ転送ﾄﾘｶﾞ
OUT TR0
AND 1110.03  ; OK_(CP1)_SFT
MOV(021) D10991 D10028  ; OKｺｰﾄﾞ, 1CH_NO_L
MOV(021) D10991 D10029  ; OKｺｰﾄﾞ, 1CH_NO_R
MOV(021) D10991 D10030  ; OKｺｰﾄﾞ, 1CH_NC_L
MOV(021) D10991 D10031  ; OKｺｰﾄﾞ, 1CH_NC_R
MOV(021) D10991 D10032  ; OKｺｰﾄﾞ, 1CH_CG_L
MOV(021) D10991 D10033  ; OKｺｰﾄﾞ, 1CH_CG_R
LD TR0
AND 1031.03  ; L_acp_(CP1)
MOV(021) D10990 D10028  ; NGｺｰﾄﾞ, 1CH_NO_L
LD TR0
AND 1032.03  ; R_acp_(CP1)
MOV(021) D10990 D10029  ; NGｺｰﾄﾞ, 1CH_NO_R
LD TR0
AND 1033.03  ; L_bcp_(CP1)
MOV(021) D10990 D10030  ; NGｺｰﾄﾞ, 1CH_NC_L
LD TR0
AND 1034.03  ; R_bcp_(CP1)
MOV(021) D10990 D10031  ; NGｺｰﾄﾞ, 1CH_NC_R
LD TR0
AND 1035.03  ; L_Cg_(CP1)
MOV(021) D10990 D10032  ; NGｺｰﾄﾞ, 1CH_CG_L
LD TR0
AND 1036.03  ; R_Cg_(CP1)
MOV(021) D10990 D10033  ; NGｺｰﾄﾞ, 1CH_CG_R
LD TR0
AND 1037.03  ; L_未測定_(CP1)
MOV(021) D10992 D10028  ; 未側ｺｰﾄﾞ, 1CH_NO_L
MOV(021) D10992 D10030  ; 未側ｺｰﾄﾞ, 1CH_NC_L
MOV(021) D10992 D10032  ; 未側ｺｰﾄﾞ, 1CH_CG_L
LD TR0
AND 1038.03  ; R_未測定_(CP1)
MOV(021) D10992 D10029  ; 未側ｺｰﾄﾞ, 1CH_NO_R
MOV(021) D10992 D10031  ; 未側ｺｰﾄﾞ, 1CH_NC_R
MOV(021) D10992 D10033  ; 未側ｺｰﾄﾞ, 1CH_CG_R

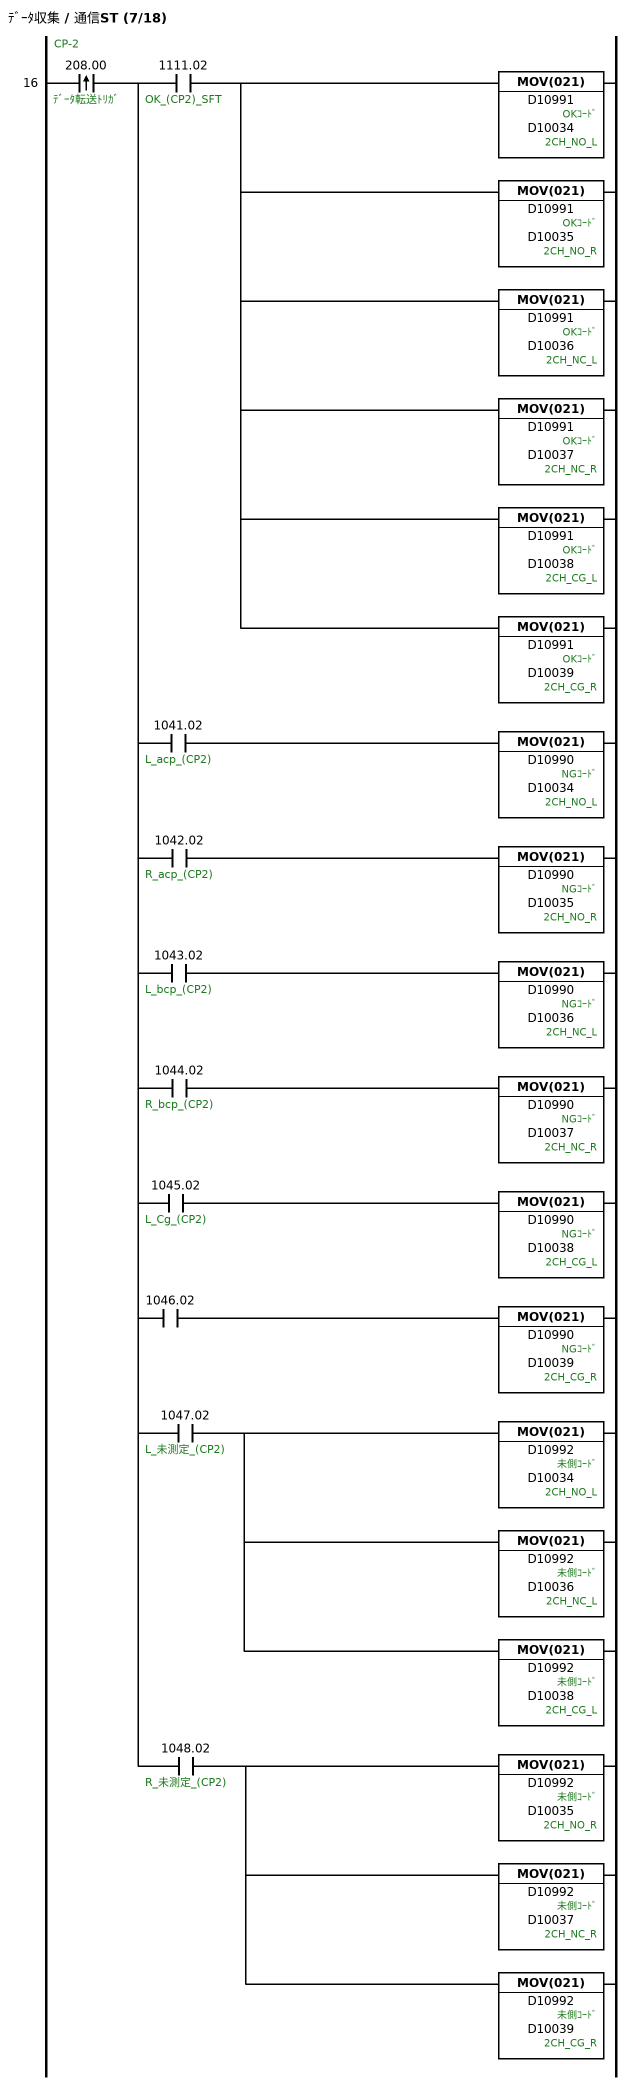
; rung 16: CP-2
@LD 208.00  ; ﾃﾞｰﾀ転送ﾄﾘｶﾞ
OUT TR0
AND 1111.02  ; OK_(CP2)_SFT
MOV(021) D10991 D10034  ; OKｺｰﾄﾞ, 2CH_NO_L
MOV(021) D10991 D10035  ; OKｺｰﾄﾞ, 2CH_NO_R
MOV(021) D10991 D10036  ; OKｺｰﾄﾞ, 2CH_NC_L
MOV(021) D10991 D10037  ; OKｺｰﾄﾞ, 2CH_NC_R
MOV(021) D10991 D10038  ; OKｺｰﾄﾞ, 2CH_CG_L
MOV(021) D10991 D10039  ; OKｺｰﾄﾞ, 2CH_CG_R
LD TR0
AND 1041.02  ; L_acp_(CP2)
MOV(021) D10990 D10034  ; NGｺｰﾄﾞ, 2CH_NO_L
LD TR0
AND 1042.02  ; R_acp_(CP2)
MOV(021) D10990 D10035  ; NGｺｰﾄﾞ, 2CH_NO_R
LD TR0
AND 1043.02  ; L_bcp_(CP2)
MOV(021) D10990 D10036  ; NGｺｰﾄﾞ, 2CH_NC_L
LD TR0
AND 1044.02  ; R_bcp_(CP2)
MOV(021) D10990 D10037  ; NGｺｰﾄﾞ, 2CH_NC_R
LD TR0
AND 1045.02  ; L_Cg_(CP2)
MOV(021) D10990 D10038  ; NGｺｰﾄﾞ, 2CH_CG_L
LD TR0
AND 1046.02
MOV(021) D10990 D10039  ; NGｺｰﾄﾞ, 2CH_CG_R
LD TR0
AND 1047.02  ; L_未測定_(CP2)
MOV(021) D10992 D10034  ; 未側ｺｰﾄﾞ, 2CH_NO_L
MOV(021) D10992 D10036  ; 未側ｺｰﾄﾞ, 2CH_NC_L
MOV(021) D10992 D10038  ; 未側ｺｰﾄﾞ, 2CH_CG_L
LD TR0
AND 1048.02  ; R_未測定_(CP2)
MOV(021) D10992 D10035  ; 未側ｺｰﾄﾞ, 2CH_NO_R
MOV(021) D10992 D10037  ; 未側ｺｰﾄﾞ, 2CH_NC_R
MOV(021) D10992 D10039  ; 未側ｺｰﾄﾞ, 2CH_CG_R

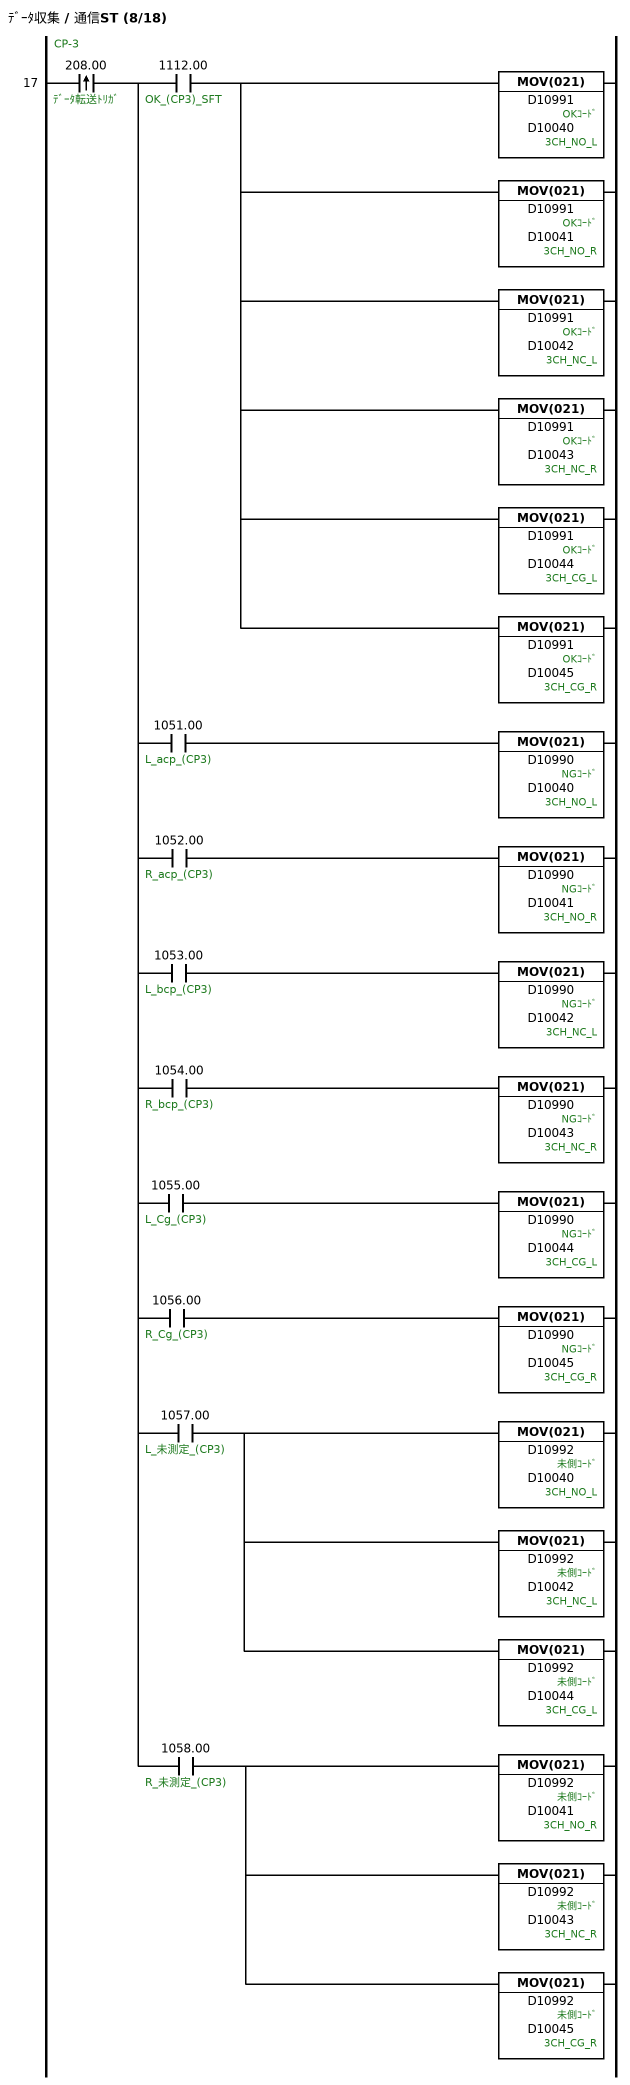
; rung 17: CP-3
@LD 208.00  ; ﾃﾞｰﾀ転送ﾄﾘｶﾞ
OUT TR0
AND 1112.00  ; OK_(CP3)_SFT
MOV(021) D10991 D10040  ; OKｺｰﾄﾞ, 3CH_NO_L
MOV(021) D10991 D10041  ; OKｺｰﾄﾞ, 3CH_NO_R
MOV(021) D10991 D10042  ; OKｺｰﾄﾞ, 3CH_NC_L
MOV(021) D10991 D10043  ; OKｺｰﾄﾞ, 3CH_NC_R
MOV(021) D10991 D10044  ; OKｺｰﾄﾞ, 3CH_CG_L
MOV(021) D10991 D10045  ; OKｺｰﾄﾞ, 3CH_CG_R
LD TR0
AND 1051.00  ; L_acp_(CP3)
MOV(021) D10990 D10040  ; NGｺｰﾄﾞ, 3CH_NO_L
LD TR0
AND 1052.00  ; R_acp_(CP3)
MOV(021) D10990 D10041  ; NGｺｰﾄﾞ, 3CH_NO_R
LD TR0
AND 1053.00  ; L_bcp_(CP3)
MOV(021) D10990 D10042  ; NGｺｰﾄﾞ, 3CH_NC_L
LD TR0
AND 1054.00  ; R_bcp_(CP3)
MOV(021) D10990 D10043  ; NGｺｰﾄﾞ, 3CH_NC_R
LD TR0
AND 1055.00  ; L_Cg_(CP3)
MOV(021) D10990 D10044  ; NGｺｰﾄﾞ, 3CH_CG_L
LD TR0
AND 1056.00  ; R_Cg_(CP3)
MOV(021) D10990 D10045  ; NGｺｰﾄﾞ, 3CH_CG_R
LD TR0
AND 1057.00  ; L_未測定_(CP3)
MOV(021) D10992 D10040  ; 未側ｺｰﾄﾞ, 3CH_NO_L
MOV(021) D10992 D10042  ; 未側ｺｰﾄﾞ, 3CH_NC_L
MOV(021) D10992 D10044  ; 未側ｺｰﾄﾞ, 3CH_CG_L
LD TR0
AND 1058.00  ; R_未測定_(CP3)
MOV(021) D10992 D10041  ; 未側ｺｰﾄﾞ, 3CH_NO_R
MOV(021) D10992 D10043  ; 未側ｺｰﾄﾞ, 3CH_NC_R
MOV(021) D10992 D10045  ; 未側ｺｰﾄﾞ, 3CH_CG_R

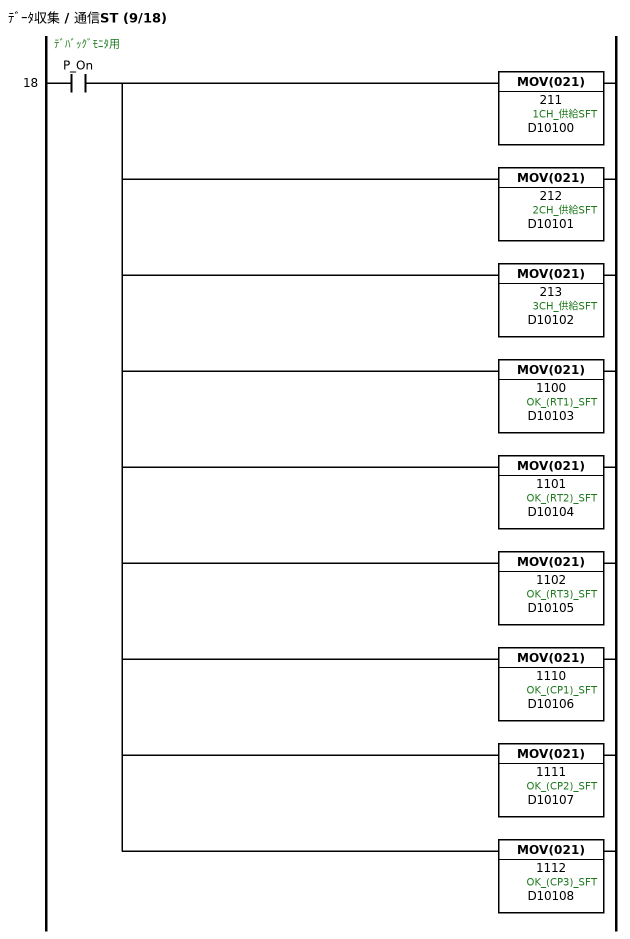
; rung 18: ﾃﾞﾊﾞｯｸﾞﾓﾆﾀ用
LD P_On
MOV(021) 211 D10100  ; 1CH_供給SFT
MOV(021) 212 D10101  ; 2CH_供給SFT
MOV(021) 213 D10102  ; 3CH_供給SFT
MOV(021) 1100 D10103  ; OK_(RT1)_SFT
MOV(021) 1101 D10104  ; OK_(RT2)_SFT
MOV(021) 1102 D10105  ; OK_(RT3)_SFT
MOV(021) 1110 D10106  ; OK_(CP1)_SFT
MOV(021) 1111 D10107  ; OK_(CP2)_SFT
MOV(021) 1112 D10108  ; OK_(CP3)_SFT

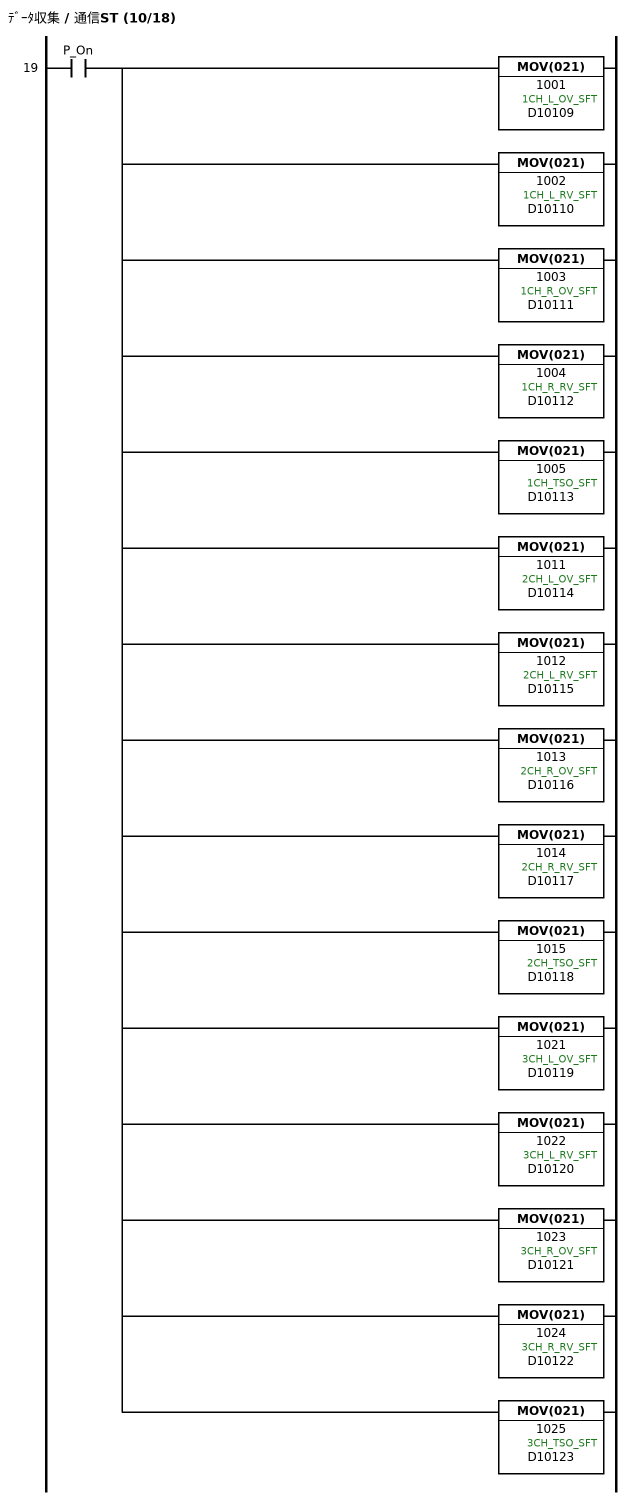
; rung 19
LD P_On
MOV(021) 1001 D10109  ; 1CH_L_OV_SFT
MOV(021) 1002 D10110  ; 1CH_L_RV_SFT
MOV(021) 1003 D10111  ; 1CH_R_OV_SFT
MOV(021) 1004 D10112  ; 1CH_R_RV_SFT
MOV(021) 1005 D10113  ; 1CH_TSO_SFT
MOV(021) 1011 D10114  ; 2CH_L_OV_SFT
MOV(021) 1012 D10115  ; 2CH_L_RV_SFT
MOV(021) 1013 D10116  ; 2CH_R_OV_SFT
MOV(021) 1014 D10117  ; 2CH_R_RV_SFT
MOV(021) 1015 D10118  ; 2CH_TSO_SFT
MOV(021) 1021 D10119  ; 3CH_L_OV_SFT
MOV(021) 1022 D10120  ; 3CH_L_RV_SFT
MOV(021) 1023 D10121  ; 3CH_R_OV_SFT
MOV(021) 1024 D10122  ; 3CH_R_RV_SFT
MOV(021) 1025 D10123  ; 3CH_TSO_SFT

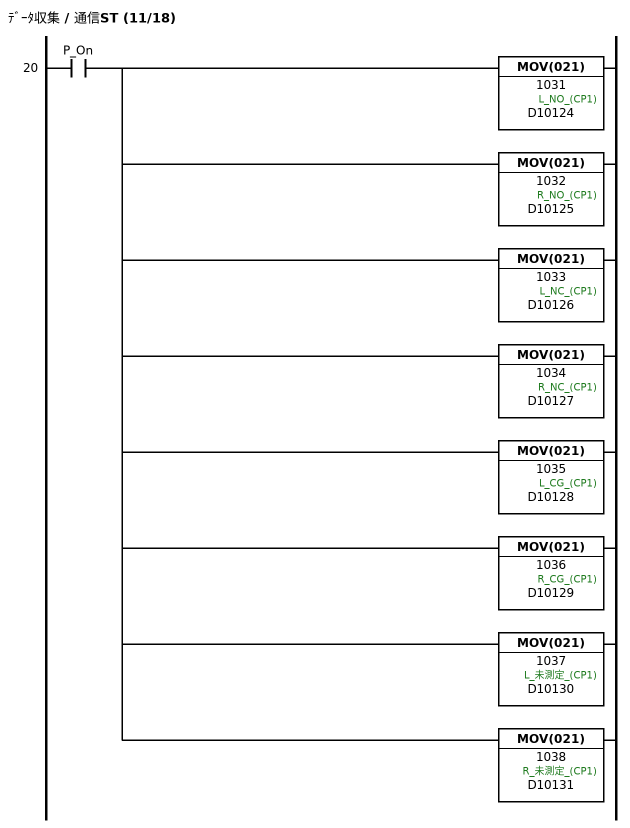
; rung 20
LD P_On
MOV(021) 1031 D10124  ; L_NO_(CP1)
MOV(021) 1032 D10125  ; R_NO_(CP1)
MOV(021) 1033 D10126  ; L_NC_(CP1)
MOV(021) 1034 D10127  ; R_NC_(CP1)
MOV(021) 1035 D10128  ; L_CG_(CP1)
MOV(021) 1036 D10129  ; R_CG_(CP1)
MOV(021) 1037 D10130  ; L_未測定_(CP1)
MOV(021) 1038 D10131  ; R_未測定_(CP1)

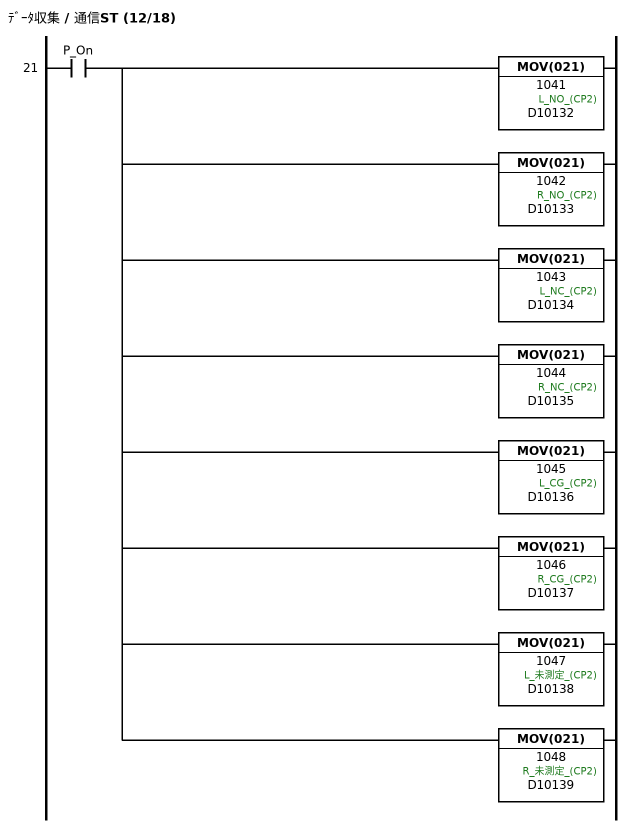
; rung 21
LD P_On
MOV(021) 1041 D10132  ; L_NO_(CP2)
MOV(021) 1042 D10133  ; R_NO_(CP2)
MOV(021) 1043 D10134  ; L_NC_(CP2)
MOV(021) 1044 D10135  ; R_NC_(CP2)
MOV(021) 1045 D10136  ; L_CG_(CP2)
MOV(021) 1046 D10137  ; R_CG_(CP2)
MOV(021) 1047 D10138  ; L_未測定_(CP2)
MOV(021) 1048 D10139  ; R_未測定_(CP2)

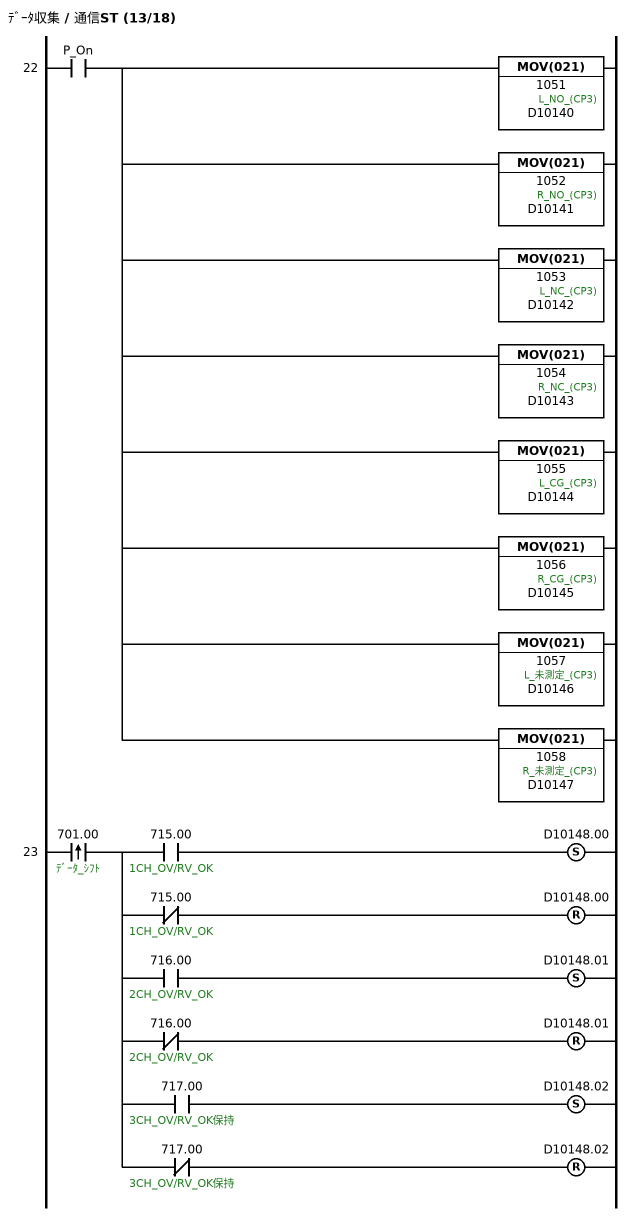
; rung 22
LD P_On
MOV(021) 1051 D10140  ; L_NO_(CP3)
MOV(021) 1052 D10141  ; R_NO_(CP3)
MOV(021) 1053 D10142  ; L_NC_(CP3)
MOV(021) 1054 D10143  ; R_NC_(CP3)
MOV(021) 1055 D10144  ; L_CG_(CP3)
MOV(021) 1056 D10145  ; R_CG_(CP3)
MOV(021) 1057 D10146  ; L_未測定_(CP3)
MOV(021) 1058 D10147  ; R_未測定_(CP3)
; rung 23
@LD 701.00  ; ﾃﾞｰﾀ_ｼﾌﾄ
OUT TR0
AND 715.00  ; 1CH_OV/RV_OK
SET D10148.00
LD TR0
ANDNOT 715.00  ; 1CH_OV/RV_OK
RSET D10148.00
LD TR0
AND 716.00  ; 2CH_OV/RV_OK
SET D10148.01
LD TR0
ANDNOT 716.00  ; 2CH_OV/RV_OK
RSET D10148.01
LD TR0
AND 717.00  ; 3CH_OV/RV_OK保持
SET D10148.02
LD TR0
ANDNOT 717.00  ; 3CH_OV/RV_OK保持
RSET D10148.02

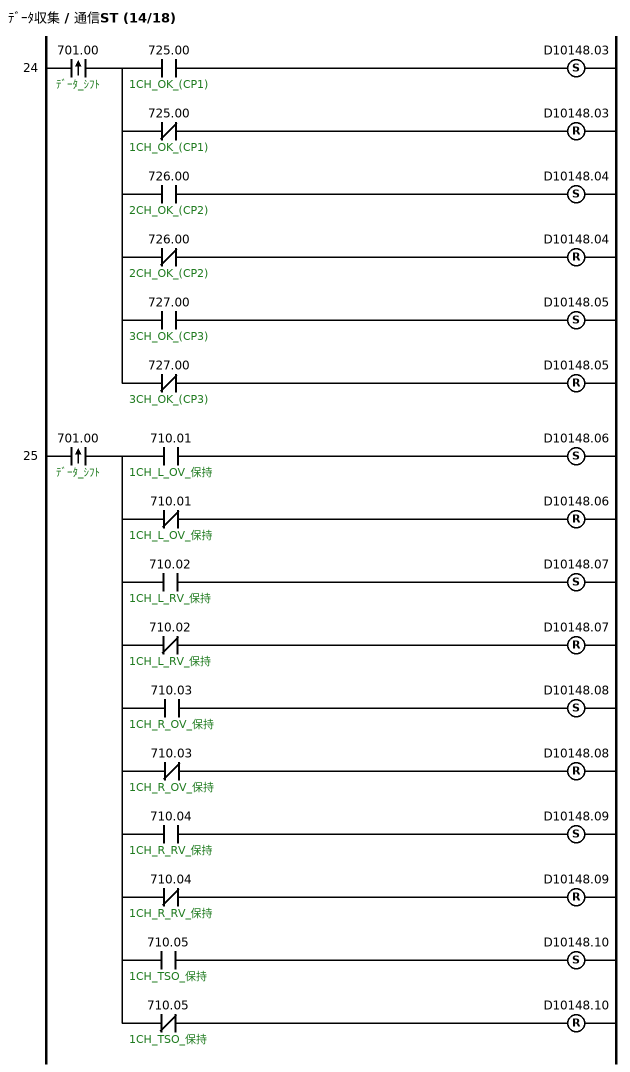
; rung 24
@LD 701.00  ; ﾃﾞｰﾀ_ｼﾌﾄ
OUT TR0
AND 725.00  ; 1CH_OK_(CP1)
SET D10148.03
LD TR0
ANDNOT 725.00  ; 1CH_OK_(CP1)
RSET D10148.03
LD TR0
AND 726.00  ; 2CH_OK_(CP2)
SET D10148.04
LD TR0
ANDNOT 726.00  ; 2CH_OK_(CP2)
RSET D10148.04
LD TR0
AND 727.00  ; 3CH_OK_(CP3)
SET D10148.05
LD TR0
ANDNOT 727.00  ; 3CH_OK_(CP3)
RSET D10148.05
; rung 25
@LD 701.00  ; ﾃﾞｰﾀ_ｼﾌﾄ
OUT TR0
AND 710.01  ; 1CH_L_OV_保持
SET D10148.06
LD TR0
ANDNOT 710.01  ; 1CH_L_OV_保持
RSET D10148.06
LD TR0
AND 710.02  ; 1CH_L_RV_保持
SET D10148.07
LD TR0
ANDNOT 710.02  ; 1CH_L_RV_保持
RSET D10148.07
LD TR0
AND 710.03  ; 1CH_R_OV_保持
SET D10148.08
LD TR0
ANDNOT 710.03  ; 1CH_R_OV_保持
RSET D10148.08
LD TR0
AND 710.04  ; 1CH_R_RV_保持
SET D10148.09
LD TR0
ANDNOT 710.04  ; 1CH_R_RV_保持
RSET D10148.09
LD TR0
AND 710.05  ; 1CH_TSO_保持
SET D10148.10
LD TR0
ANDNOT 710.05  ; 1CH_TSO_保持
RSET D10148.10

